(* IEC 61131-3 sources: elnaProjects/ElpcLogic/PomarKc7Changed/build_USO_ecl (part 8) *)

  IF isRunning THEN
  	Signaling := inSignaling;
  	SignalingTP := _signalingTp.Q;
  ELSE
  	Signaling := 0;
  	SignalingTP := 0;
  END_IF;

  IF NOT Remont AND NOT Check THEN
  	_signalingTp(in := Signaling, PT := T#1s);
  ELSE
  	_signalingTp(in := FALSE);
  END_IF;

  status :=  SHL(BYTE_TO_DWORD(source_for_Status), 29)
  			OR SHL(BYTE_TO_DWORD(cmd_for_Status), 26)
  			OR SHL(BYTE_TO_DWORD(command_error_for_Status), 23)
  			OR SHL(BOOL_TO_DWORD(OpcCommandsDisabled ), 21)
  			OR SHL(BOOL_TO_DWORD(Signaling), 16)
  			OR SHL(BOOL_TO_DWORD(RunOnStart ), 15)
  			OR SHL(BOOL_TO_DWORD(remont), 6)
  			OR SHL(BOOL_TO_DWORD(Check), 5)
  			OR SHL(BOOL_TO_DWORD(hasError), 4)
  			OR SHL(BOOL_TO_DWORD(SignalingTP), 3)
  			OR SHL(BOOL_TO_DWORD(CanRun), 2)
  			OR SHL(BOOL_TO_DWORD(isEnded), 1)
  			OR BOOL_TO_DWORD(isRunning);
END_FUNCTION_BLOCK

FUNCTION_BLOCK fb_BaseAlgoritm
  VAR_IN_OUT
    StrAlg : struct_Alg;
  END_VAR
  VAR
    _sunpackerCommand : fb_sunpackerCommand;
    source : BYTE;
    cmd : BYTE;
    lastCmd : BYTE;
    source_for_Status : BYTE;
    cmd_for_Status : BYTE;
    command_error_for_Status : BYTE;
    resetCmdTimer : TON;
    resetCmdTimerPriznak : BOOL;
  END_VAR

  StrAlg.CanRun := StrAlg.inCanRun;
  StrAlg.hasError := StrAlg.inHasError OR (command_error_for_Status <> 0);
  StrAlg.isEnded := StrAlg.inEnded;

  StrAlg.OpcCommandsDisabled := StrAlg.inOpcCommandsDisabled;

  (* ---- Если управление с ВУ заблокировано, то передаем команду из алгоритма ---- *)
  IF StrAlg.inOpcCommandsDisabled THEN
  	StrAlg.inCommand := StrAlg.inCommand_Alg;
  ELSE (* иначе передаем команду с АРМа*)
  	StrAlg.inCommand := StrAlg.inCommand_ARM;
  END_IF;

  _sunpackerCommand(command := StrAlg.inCommand);
  	source := _sunpackerCommand.source;
  	cmd := _sunpackerCommand.cmd;

  IF cmd <> 0 AND lastCmd <> cmd AND (((NOT StrAlg.opcCommandsDisabled) AND source > 0) OR source = 0) then
  	CASE BYTE_TO_INT(cmd) OF
  		(*cmdRun*) 1: 	IF (StrAlg.CanRun) THEN
  					StrAlg.isRuning := TRUE;
  					StrAlg.isEnded := FALSE;
  					StrAlg.hasError 	:= FALSE;

  					cmd_for_Status := cmd;
  					source_for_Status := source;
  					command_error_for_Status := 0;
  				ELSE
  					StrAlg.isRuning := FALSE;
  					StrAlg.isEnded := FALSE;
  					StrAlg.hasError 	:= FALSE;

  					cmd_for_Status := 0;
  					source_for_Status := source;
  					command_error_for_Status := cmd;
  				END_IF;
  		(*cmdReset*) 2: 	StrAlg.isRuning := FALSE;
  				StrAlg.isEnded := FALSE;
  				StrAlg.hasError 	:= FALSE;
  				cmd_for_Status := cmd;
  				source_for_Status := source;
  				command_error_for_Status := 0;
  	END_CASE;
  	resetCmdTimer(IN := false);
  	resetCmdTimerPriznak := TRUE;
  END_IF;
  lastCmd := cmd;

  resetCmdTimer(IN := resetCmdTimerPriznak, PT := T#5S);
  IF resetCmdTimer.Q THEN
  	resetCmdTimerPriznak := FALSE;
  	source_for_Status := 0;
  	cmd_for_Status := 0;
  	command_error_for_Status := 0;
  END_IF;

  StrAlg.status :=  SHL(BYTE_TO_DWORD(source_for_Status), 29)
  			OR SHL(BYTE_TO_DWORD(cmd_for_Status), 26)
  			OR SHL(BYTE_TO_DWORD(command_error_for_Status), 23)
  			OR SHL(BOOL_TO_DWORD(StrAlg.OpcCommandsDisabled ), 21)
  			OR SHL(BOOL_TO_DWORD(StrAlg.hasError),4)
  			OR SHL(BOOL_TO_DWORD(StrAlg.CanRun),2)
  			OR SHL(BOOL_TO_DWORD(StrAlg.isEnded),1)
  			OR BOOL_TO_DWORD(StrAlg.isRuning);
END_FUNCTION_BLOCK

FUNCTION_BLOCK fb_Switch
  VAR_INPUT
    statOn : BOOL;
    statOff : BOOL;
    statOn_reliability : BOOL;
    statOff_reliability : BOOL;
  END_VAR
  VAR_IN_OUT
    StrSw : struct_Switch;
  END_VAR
  VAR_INPUT
    inNs : TYPE_ReliableBit;
    inAccident : TYPE_ReliableBit;
    inAuto : TYPE_ReliableBit;
    inManual : TYPE_ReliableBit;
    inLocal : TYPE_ReliableBit;
    inDistance : TYPE_ReliableBit;
    inErrorPowerOff : TYPE_ReliableBit;
    inErrorBlock : TYPE_ReliableBit;
    inBreakCmdOn : TYPE_ReliableBit;
    inBreakCmdOff : TYPE_ReliableBit;
  END_VAR
  VAR
    onInit : BOOL          := FALSE;
    _statOn : BOOL;
    _statOff : BOOL;
    lastOnStatus : BYTE;
    cmd : BYTE;
    source : BYTE;
    lastCmd : BYTE;
    source_for_Status : BYTE;
    cmd_for_Status : BYTE;
    command_error_for_Status : BYTE;
    _sunpackerCommand : fb_sunpackerCommand;
    _statusDualInput : TYPE_statusDualInput;
    _commandDualInput : TYPE_commandDualInput;
    _commandErrorTimer : BOOL;
    resetErrorTimer : BOOL;
    getSdvig : BOOL;
    _changWithoutCommand : BOOL;
    errorCMDTimer : TON;
    sdvigReset : TON;
    _errorReset : TON;
    outputsSets : TOF;
  END_VAR
  VAR_IN_OUT
    cmdOn : BOOL;
    cmdOff : BOOL;
  END_VAR

  IF NOT onInit THEN
  IF StrSw.ISVALIDREF_cmdOn XOR StrSw.ISVALIDREF_cmdOff THEN
  	IF 	StrSw.ISVALIDREF_cmdOn THEN
  		lastCmd:= 2; (*baseCmdOff*)
  	ELSE
  		lastCmd:= 1; (*baseCmdOn*)
  	END_IF;
  END_IF;
  onInit:=TRUE;
  END_IF;

  (* ---- Если управление с ВУ заблокировано, то в ИМ передаем команду из алгоритма ---- *)
  IF StrSw.inOpcCommandsDisabled THEN
  	StrSw.inCommand := StrSw.inCommand_Alg;
  ELSE (* иначе передаем команду с АРМа*)
  	StrSw.inCommand := StrSw.inCommand_ARM;
  END_IF;

  (* ---- Формирование состояния механизма ---- *)

  IF (StrSw.ISVALIDREF_statOn) OR (StrSw.ISVALIDREF_statOff) THEN
  	IF (StrSw.ISVALIDREF_statOn) AND (StrSw.ISVALIDREF_statOff) THEN
  	StrSw.reliability:= statOn_reliability AND statOff_reliability;
  		_statOn  := statOn;
  		_statOff := statOff;
  	ELSIF (StrSw.ISVALIDREF_statOn) THEN
                       StrSw.reliability:= statOn_reliability;
  		_statOn  := statOn;
  		_statOff := NOT statOn;
  	ELSIF (StrSw.ISVALIDREF_statOff) THEN
  		 StrSw.reliability:= statOff_reliability;
  		_statOn  := NOT statOff;
  		_statOff :=statOff;
  	END_IF;

  	IF StrSw.reliability THEN
  		IF _statOn AND NOT _statOff 		THEN 	StrSw.onStatus := _statusDualInput.STATUS_ON;
  		ELSIF _statOff AND NOT _statOn 	THEN 	StrSw.onStatus := _statusDualInput.Status_OFF;
  		ELSIF NOT _statOn AND NOT _statOff 	THEN 	StrSw.onStatus := _statusDualInput.STATUS_TRANSITIONAL;
  		ELSE					StrSw.onStatus := _statusDualInput.STATUS_ERROR;
                      END_IF;

  	ELSE
  		StrSw.onStatus := _statusDualInput.STATUS_NOTDEFINED;

  	END_IF;
  ELSE
  	CASE BYTE_TO_INT(lastCmd) OF
  		(*baseCmdOn*) 1: StrSw.onStatus  := _statusDualInput.STATUS_ON;
  		(*baseCmdOff*) 2: StrSw.onStatus  := _statusDualInput.STATUS_OFF;

  	ELSE
  		 StrSw.onStatus := _statusDualInput.STATUS_NOTDEFINED;

  	END_CASE;
  END_IF;

  StrSw.Accident := inAccident.value AND inAccident.reliability;
  StrSw.Ns := inNs.value AND inNs.reliability;
  StrSw.Auto := inAuto.value AND inAuto.reliability;
  StrSw.Manual := inManual.value AND inManual.reliability;
  StrSw.Local := inLocal.value AND inLocal.reliability;
  StrSw.Distance := inDistance.value AND inDistance.reliability;
  StrSw.ErrorPowerOff := inErrorPowerOff.value AND inErrorPowerOff.reliability;
  StrSw.ErrorBlock := inErrorBlock.value AND inErrorBlock.reliability;
  StrSw.OpcCommandsDisabled := StrSw.inOpcCommandsDisabled;

  (* ---- Формирование признака сдвига ---- *)
  getSdvig := FALSE;
  IF (StrSw.ISVALIDREF_cmdOn OR StrSw.ISVALIDREF_cmdOff) AND NOT StrSw.Local THEN
  	IF NOT (StrSw.CmdOn OR StrSw.CmdOff) THEN
                       IF (lastOnStatus <> StrSw.onStatus AND
  		(StrSw.onStatus <> _statusDualInput.STATUS_NOTDEFINED AND
                       StrSw.onStatus <> _statusDualInput.STATUS_ERROR)     AND
  		(lastOnStatus <> _statusDualInput.STATUS_NOTDEFINED   AND
                       lastOnStatus <> _statusDualInput.STATUS_ERROR))
                      THEN
  			getSdvig   := TRUE;
  		END_IF;
  	END_IF;
  END_IF;

  IF getSdvig THEN StrSw.sdvig:= TRUE; END_IF;

  sdvigReset(IN:=StrSw.sdvig, PT:=T#15S);

  IF sdvigReset.Q THEN StrSw.sdvig:=FALSE; END_IF;

  lastOnStatus := StrSw.onStatus;

  (* ---- Распаковка команды ---- *)
  _sunpackerCommand(command := StrSw.inCommand);
  	cmd := _sunpackerCommand.cmd;
  	source := _sunpackerCommand.source;

  (* ---- Обработка команды ---- *)
  IF cmd <> 0 AND lastCmd <> cmd and (((NOT StrSw.opcCommandsDisabled) AND source > 0) OR source = 0) then
  	CASE BYTE_TO_INT(cmd) OF
  	(*cmd_open*) 1 :
  			IF  StrSw.ISVALIDREF_cmdOn THEN StrSw.CmdOn := TRUE;
  				IF StrSw.ISVALIDREF_cmdOff THEN StrSw.CmdOff := FALSE; END_IF;
  			ELSIF  StrSw.ISVALIDREF_cmdOff THEN StrSw.CmdOff := FALSE;  END_IF;
                                lastCmd := cmd;
  			errorCMDTimer(IN := false);
  			_commandErrorTimer := true;
  			StrSw.lastCmdIsOn := true;
  	(*cmd_close*) 2 :
  			IF StrSw.ISVALIDREF_cmdOff THEN StrSw.CmdOff := TRUE;
  				IF StrSw.ISVALIDREF_cmdOn THEN StrSw.CmdOn := FALSE; END_IF;
  			ELSIF StrSw.ISVALIDREF_cmdOn THEN StrSw.CmdOn := FALSE; END_IF;
                                lastCmd := cmd;
  			errorCMDTimer(IN := false);
  			_commandErrorTimer := true;
  			StrSw.lastCmdIsOn := false;
  	(*cmd_reset*) 3 :    IF StrSw.ISVALIDREF_statOn OR StrSw.ISVALIDREF_statOff THEN
  			StrSw.CmdOn := FALSE;
  			StrSw.CmdOff := FALSE;
                                lastCmd :=0;
  			_commandErrorTimer := false;
  			StrSw.lastCmdIsOn := false;
                                 END_IF;
  	END_CASE;
  	source_for_Status := source;
  	cmd_for_Status := cmd;
  	command_error_for_Status := 0;
  END_IF;

  errorCMDTimer(In := _commandErrorTimer, PT :=T#10s);

  (* ---- алгоритм  для команды ВКЛючить ---- *)
  IF (StrSw.onStatus = _statusDualInput.STATUS_ON) and StrSw.lastCmdIsOn then
  	IF StrSw.ISVALIDREF_cmdOn AND StrSw.ISVALIDREF_cmdOff then  StrSw.cmdOn := false; END_IF;

  	 errorCMDTimer(In := false);
  	 _commandErrorTimer := false;
  	 cmd_for_Status := 0;
  	 source_for_Status := 0;
  END_IF;

  (* ---- off ---- *)
  IF (StrSw.onStatus = _statusDualInput.STATUS_OFF) and (NOT StrSw.lastCmdIsOn) then
  	IF StrSw.ISVALIDREF_cmdOn AND StrSw.ISVALIDREF_cmdOff then  StrSw.cmdOff := false; END_IF;

  	 errorCMDTimer(In := false);
  	 _commandErrorTimer := false;
  	 cmd_for_Status := 0;
  	 source_for_Status := 0;
  END_IF;

  (* ---- ошибка исполнения команды ---- *)
  if errorCMDTimer.Q and (cmd_for_Status <> 0) then
  	command_error_for_Status :=  cmd_for_Status;
  	_commandErrorTimer := false;
  	StrSw.CmdOn := false;
  	StrSw.CmdOff := false;
  	lastCmd := 0;
  end_if;

  (* ---- сброс ошибки команды ---- *)
  StrSw.CommandFault := command_error_for_Status <> 0;
  _errorReset(IN := command_error_for_Status <> 0, PT := T#5S);
  IF _errorReset.Q THEN
  	cmd_for_Status := 0;
  	source_for_Status := 0;
  	command_error_for_Status := 0;
  END_IF;

  outputsSets(in := (StrSw.ISVALIDREF_cmdOn and StrSw.cmdOn ) OR (StrSw.ISVALIDREF_cmdOff and StrSw.cmdOff), PT := T#2S);
  	IF NOT outputsSets.Q THEN
  		StrSw.BreakCmdOn := inBreakCmdOn._inversed AND
                      inBreakCmdOn.reliability AND StrSw.ISVALIDREF_inBreakCmdOn;

  		StrSw.BreakCmdOff := inBreakCmdOff._inversed
                      AND inBreakCmdOff.reliability AND StrSw.ISVALIDREF_inBreakCmdOff;
  	END_IF;

  cmdOn := StrSw.cmdOn;
  cmdOff:= StrSw.cmdOff;

  (* ---- формирование зашифрованного статуса для АРМа ---- *)
  StrSw.status := shl(BYTE_TO_DWORD(source_for_Status), 29)
  		OR shl(BYTE_TO_DWORD(cmd_for_Status), 26)
  		OR shl(BYTE_TO_DWORD(command_error_for_Status), 23)
  		OR shl(bool_to_DWORD(StrSw.sdvig), 22)
  		OR shl(bool_to_DWORD(StrSw.OpcCommandsDisabled), 21)
                      OR shl(bool_to_DWORD(StrSw.lastCmdIsOn), 14)
                      OR shl(BOOL_TO_DWORD(StrSw.BreakCmdOff), 13)
  		OR shl(BOOL_TO_DWORD(StrSw.BreakCmdOn), 12)
  		OR shl(BOOL_TO_DWORD(StrSw.ErrorBlock), 11)
  		OR shl(BOOL_TO_DWORD(StrSw.ErrorPowerOff), 10)
  		OR shl(BOOL_TO_DWORD(StrSw.Manual), 8)
  		OR shl(BOOL_TO_DWORD(StrSw.Auto), 7)
  		OR shl(BOOL_TO_DWORD(StrSw.Distance), 6)
  		OR shl(BOOL_TO_DWORD(StrSw.Local), 5)
  		OR shl(BOOL_TO_DWORD(StrSw.Ns), 4)
                  	OR shl(BOOL_TO_DWORD(StrSw.Accident ),3)
  		OR BYTE_TO_DWORD(StrSw.onStatus);
END_FUNCTION_BLOCK

FUNCTION_BLOCK fb_singleOutput
  VAR_IN_OUT
    signal : BOOL;
    str_SO : struct_singleOutput;
  END_VAR
  VAR
    pulseTimer : TON;
    resetCmdTimer : TON;
    TON_Command : TON;
    source : BYTE;
    cmd : BYTE;
    lastCmd : BYTE;
    source_for_Status : BYTE;
    cmd_for_Status : BYTE;
    command_error_for_Status : BYTE;
    pulseTimerPriznak : BOOL;
    resetCmdTimerPriznak : BOOL;
    _sunpackerCommand : fb_sunpackerCommand;
  END_VAR

  str_SO.OpcCommandsDisabled := str_SO.inOpcCommandsDisabled;

  (* ---- Если управление с ВУ заблокировано, то передаем команду из алгоритма ---- *)
  IF str_SO.inOpcCommandsDisabled THEN
  	str_SO.inCommand := str_SO.inCommand_Alg;
  ELSE (* иначе передаем команду с АРМа*)
  	str_SO.inCommand := str_SO.inCommand_ARM;
  END_IF;

  (*Распаковка команды*)
  _sunpackerCommand(command := str_SO.inCommand);
  	cmd := _sunpackerCommand.cmd;
  	source := _sunpackerCommand.source;

  (*Обработка команды*)
  IF cmd <> 0 AND lastCmd <> cmd and (((NOT str_SO.OpcCommandsDisabled) AND source > 0) OR source = 0) then
  	CASE BYTE_TO_INT(cmd) OF
  	(*cmd_on*) 1 :
  			str_SO.Q := TRUE;
  			pulseTimer(IN := FALSE);
  			pulseTimerPriznak := FALSE;
  			resetCmdTimer(IN := FALSE);
  			resetCmdTimerPriznak := TRUE;
  	(*cmd_off*) 2 :
  			str_SO.Q := FALSE;
  			pulseTimer(IN := FALSE);
  			pulseTimerPriznak := FALSE;
  			resetCmdTimer(IN := FALSE);
  			resetCmdTimerPriznak := TRUE;
  	(*cmd_pulse*) 3 :
  			str_SO.Q := TRUE;
                                pulseTimer(IN := FALSE);
                                pulseTimerPriznak := TRUE;
  			resetCmdTimer(IN := FALSE);
                                resetCmdTimerPriznak := FALSE;
  	END_CASE;
  	source_for_Status := source;
  	cmd_for_Status := cmd;
  	command_error_for_Status := 0;
  END_IF;
  lastCmd := cmd;

  pulseTimer(IN := pulseTimerPriznak, PT := str_SO.wait_time);
  pulseTimer();
  IF pulseTimer.Q THEN
  	pulseTimer(IN := FALSE);
  	pulseTimerPriznak := FALSE;

  	str_SO.Q := FALSE;

  	source_for_Status := 0;
  	cmd_for_Status := 0;
  	command_error_for_Status := 0;
  END_IF;

  resetCmdTimer(IN := resetCmdTimerPriznak, PT := T#10S);
  resetCmdTimer();
  IF resetCmdTimer.Q THEN
  	resetCmdTimer(IN := FALSE);
  	resetCmdTimerPriznak := FALSE;

  	source_for_Status := 0;
  	cmd_for_Status := 0;
  	command_error_for_Status := 0;
  END_IF;

  signal:= str_SO.Q;

  (*TON_Command(IN:= (inCommand <> 0) AND (source = 0), PT:= T#2S);*)
      (*IF TON_Command.Q THEN*)
          (*inCommand := 0;*)
      (*END_IF;*)
  str_SO.status :=                           shl(BYTE_TO_DWORD(source_for_Status), 29)
  				OR shl(BYTE_TO_DWORD(cmd_for_Status), 26)
  				OR shl(BYTE_TO_DWORD(command_error_for_Status), 23)
  				OR shl(BOOL_TO_DWORD(str_SO.OpcCommandsDisabled), 21)
  				OR BOOL_TO_DWORD(str_SO.Q);
END_FUNCTION_BLOCK

FUNCTION_BLOCK proc_IM
  VAR
    fb_Kran1 : fb_Kran;
    fb_Kran2 : fb_Kran;
    fb_Kran3 : fb_Kran;
    fb_Kran3b : fb_Kran;
    fb_Kran4 : fb_Kran;
    fb_Kran5 : fb_Kran;
    fb_Kran6 : fb_Kran;
    fb_nu1 : fb_OilPump;
    fb_nu2 : fb_OilPump;
    fb_pns : fb_Switch;
    fb_v1_Avom : fb_Switch;
    fb_v2_Avom : fb_Switch;
    fb_v3_Avom : fb_Switch;
    fb_v4_Avom : fb_Switch;
    fb_TEN_kollectora : fb_Switch;
    fb_KaloriferAVOM : fb_Switch;
    fb_CMN : fb_Switch;
    fb_TEN_MB : fb_Switch;
    fb_mv : fb_SectionSwitch;
    fb_PLC_Control : fb_meandr;
  END_VAR
  VAR_EXTERNAL
    di : DiConfig;
    od : DOconfig;
    IM : ImConfig;
  END_VAR
  VAR
    fb_dP_maslo_gaz_Less100 : fb_singleSignal;
    fb_dp_kran1_Less100 : fb_singleSignal;
    fb_QF1_on : fb_singleSignal;
    fb_QF2_on : fb_singleSignal;
    fb_QF23_on : fb_singleSignal;
    fb_QF4_QF5_on : fb_singleSignal;
    fb_QF6_QF7_on : fb_singleSignal;
    fb_QF8_QF9_on : fb_singleSignal;
    fb_QF10_QF11_on : fb_singleSignal;
    fb_QF12_QF13_on : fb_singleSignal;
    fb_QF14_QF15_on : fb_singleSignal;
    fb_QF22_on : fb_singleSignal;
    fb_NS_G1_G2 : fb_singleSignal;
    fb_NS_G3_G4 : fb_singleSignal;
    fb_NS_G15_G16 : fb_singleSignal;
    fb_NS_G17 : fb_singleSignal;
    fb_NS_G5_G6 : fb_singleSignal;
    fb_NS_G7_G8 : fb_singleSignal;
    fb_NS_G18_G19 : fb_singleSignal;
    fb_NS_G10_G11 : fb_singleSignal;
    fb_NS_G13_G14 : fb_singleSignal;
    fb_Vozbud_neispr_tsepey_upr_AVR_pit : fb_singleSignal;
    fb_Vozbud_gotovnost : fb_singleSignal;
    fb_Vozbud_neispravnost : fb_singleSignal;
    fb_SHAVR1_v_rabote : fb_singleSignal;
    fb_SHAVR2_v_rabote : fb_singleSignal;
    fb_Avariinoe_otkluch_vikluchatelya : fb_singleSignal;
    fb_Assinhronnii_hod_peregruzka : fb_singleSignal;
    fb_SHU_v_GPA_vkluch : fb_singleSignal;
    fb_SHP_v_GPA_vkluch : fb_singleSignal;
    fb_Uroven_masla_akkum : fb_singleSignal;
    fb_NKU1_GPA_on : fb_singleSignal;
    fb_NKU2_GPA_on : fb_singleSignal;
    fb_AO_KC_ot_SHKS : fb_singleSignal;
    fb_AO_GPA_ot_SHU : fb_singleSignal;
    fb_BEAO_srabotal : fb_singleSignal;
    fb_Chastotny_pusk : fb_singleSignal;
    fb_Neuspesh_chastotny_pusk : fb_singleSignal;
    fb_Rezhim_ruchnogo_regulirovaniya : fb_singleSignal;
    fb_Razreshenie_zagruzki_dvig : fb_singleSignal;
    fb_Osnovnoy_regul_off : fb_singleSignal;
    fb_Voltage_sekcii_norm : fb_singleSignal;
    fb_Reactorny_pusk : fb_singleSignal;
    fb_NO_GPA_ot_SHU : fb_singleSignal;
    fb_AO_GPA_ot_PRU : fb_singleSignal;
    fb_Nalichie_BP1 : fb_singleSignal;
    fb_Nalichie_BP2 : fb_singleSignal;
    fb_Nalichie_BP3 : fb_singleSignal;
    fb_Nalichie_BP4 : fb_singleSignal;
    fb_Nalichie_BP5 : fb_singleSignal;
    fb_Nalichie_BP6 : fb_singleSignal;
    fb_Nalichie_BP7_BP8 : fb_singleSignal;
    fb_Nalichie_BP9_BP10 : fb_singleSignal;
    fb_Nalichie_cepei_upravlen_mv : fb_singleSignal;
    fb_Nalichie_220BEAO : fb_singleSignal;
    fb_Nalichie_per_220_na_vhode : fb_singleSignal;
    fb_Nalichie_post_220_na_vhode : fb_singleSignal;
    fb_Nalichie_BP11 : fb_singleSignal;
    fb_Nalichie_BP12 : fb_singleSignal;
    fb_Dver_SHU_pered_otkrita : fb_singleSignal;
    fb_Dver_SHU_zad_otkrita : fb_singleSignal;
    fb_EO_GPA_ot_knopki_SHU : fb_singleSignal;
    fb_EO_EGPA_ot_PRY : fb_singleSignal;
    fb_Synchroniz_rezhima_K1 : fb_singleSignal;
    fb_Potok_ms_posle_AVOM : fb_singleSignal;
    fb_Avary_EGPA : fb_singleOutput;
    fb_U_lamp_SHU : fb_singleOutput;
    fb_AO_knopka_ind : fb_singleOutput;
    fb_Pusk : fb_singleOutput;
    fb_Stop_SHUP : fb_singleOutput;
    fb_NO_fonar : fb_singleOutput;
    fb_PC_fonar : fb_singleOutput;
    fb_AC_fonar : fb_singleOutput;
    fb_Kr1_smazka : fb_singleOutput;
    fb_Kr2_smazka : fb_singleOutput;
    fb_Kr4_open_from_alg : fb_singleOutput;
    fb_Synch_rej_K1 : fb_singleOutput;
    fb_Rabota_EGPA : fb_singleOutput;
    fb_Neispr_EGPA : fb_singleOutput;
  END_VAR

  (* Циклический опрос. ИМ *)

  (* GPIO *)
  fb_PLC_Control(output:=od.gpio_out.bits[0]);

  (* Кран 1 *)
  fb_Kran1(statOn := di.di_20.bits[5]._inversed,
           statOff := di.di_20.bits[4]._inversed,
           inSo := di.di_16.bits[0], inSz := di.di_16.bits[1],
           cmdOn:=od.do_0.bits[0], cmdOff:=od.do_0.bits[1],
           strKr:= IM.Kran1  );

  (* Кран 2 *)
  fb_Kran2(statOn := di.di_21.bits[0]._inversed,
           statOff := di.di_20.bits[7]._inversed,
           inSo := di.di_16.bits[2], inSz := di.di_16.bits[3],
           cmdOn:=od.do_0.bits[2], cmdOff:=od.do_0.bits[3],
           strKr:= IM.Kran2  );

  (* Кран 3 *)
  fb_Kran3(statOn := di.di_0.bits[5]._inversed,
           statOff := di.di_0.bits[4]._inversed,
           inSo := di.di_16.bits[4], inSz := di.di_16.bits[5],
           cmdOn:=od.do_0.bits[4], cmdOff:=od.do_0.bits[5],
           strKr:= IM.Kran3  );

  (* Кран 3b *)
  fb_Kran3b(statOn := di.di_0.bits[7]._inversed,
           statOff := di.di_0.bits[6]._inversed,
           inSo := di.di_16.bits[6], inSz := di.di_16.bits[7],
           cmdOn:=od.do_0.bits[6], cmdOff:=od.do_0.bits[7],
           strKr:= IM.Kran3b  );

  (* Кран 4 *)
  fb_Kran4(statOn := di.di_1.bits[1]._inversed,
           statOff := di.di_1.bits[0]._inversed,
           inSo := di.di_17.bits[0], inSz := di.di_17.bits[1],
           cmdOn:=od.do_0.bits[8], cmdOff:=od.do_0.bits[9],
           strKr:= IM.Kran4  );

  (* Кран 5 *)
  fb_Kran5(statOn := di.di_1.bits[3]._inversed,
           statOff := di.di_1.bits[2]._inversed,
           inSo := di.di_17.bits[2], inSz := di.di_17.bits[3],
           cmdOn:=od.do_0.bits[10], cmdOff:=od.do_0.bits[11],
           strKr:= IM.Kran5  );

  (* Кран 6НР *)
  fb_Kran6(statOn := di.di_1.bits[5]._inversed,
           statOff := di.di_1.bits[4]._inversed,
           inSo := di.di_17.bits[4], inSz := di.di_17.bits[5],
           cmdOn:=od.do_0.bits[12], cmdOff:=od.do_0.bits[13],
           strKr:= IM.Kran6  );

  (*  НУ1 Насос уплотнения *)
  fb_nu1(statOn := di.di_5.bits[1].value, statOff := di.di_5.bits[1]._inversed,
           cmdOn:=od.do_1.bits[4], cmdOff:=od.do_1.bits[5],
           StrSw:= IM.nu1  );

  (*  НУ2 Насос уплотнения *)
  fb_nu2(statOn := di.di_5.bits[2].value, statOff := di.di_5.bits[2]._inversed,
           cmdOn:=od.do_1.bits[6], cmdOff:=od.do_1.bits[7],
           StrSw:= IM.nu2  );

  (*  ПНС Насос смазки *)
  fb_pns(statOn := di.di_5.bits[0].value, statOff := di.di_5.bits[0]._inversed,
           cmdOn:=od.do_1.bits[0], cmdOff:=od.do_1.bits[1],
           StrSw:= IM.pns  );

  (*  В1 АВОМ вентилятор охлаждения *)
  fb_v1_Avom(statOn := di.di_5.bits[3].value, statOff := di.di_5.bits[3]._inversed,
           cmdOn:=od.do_1.bits[8], cmdOff:=od.do_1.bits[9],
           StrSw:= IM.v1_Avom  );

  (*  В2 АВОМ вентилятор охлаждения *)
  fb_v2_Avom(statOn := di.di_5.bits[4].value, statOff := di.di_5.bits[4]._inversed,
           cmdOn:=od.do_1.bits[10], cmdOff:=od.do_1.bits[11],
           StrSw:= IM.v2_Avom  );

  (*  В3 АВОМ вентилятор охлаждения *)
  fb_v3_Avom(statOn := di.di_5.bits[5].value, statOff := di.di_5.bits[5]._inversed,
           cmdOn:=od.do_1.bits[12], cmdOff:=od.do_1.bits[13],
           StrSw:= IM.v3_Avom  );

  (*  В4 АВОМ вентилятор охлаждения *)
  fb_v4_Avom(statOn := di.di_5.bits[6].value, statOff := di.di_5.bits[6]._inversed,
           cmdOn:=od.do_1.bits[14], cmdOff:=od.do_1.bits[15],
           StrSw:= IM.v4_Avom  );

  (*  МВ масляный выключатель *)
  fb_mv(statOn := di.di_7.bits[0].value, statOff := di.di_20.bits[3].value,
           basketRolledin:= di.di_7.bits[2], basketRolledout:= di.di_7.bits[2],
           cmdOn:=od.do_4.bits[6] , cmdOff:=od.do_4.bits[7],
           StrSw:= IM.mv  );

  (* Тен коллектора *)
  fb_TEN_kollectora(statOn := di.di_10.bits[1].value, statOff := di.di_10.bits[1]._inversed,
           cmdOn:=od.do_2.bits[6], cmdOff:=od.do_2.bits[6],
           StrSw:= IM.TEN_kollectora  );

  (* Калорифер АВОМ *)
  fb_KaloriferAVOM(statOn := di.di_10.bits[2].value, statOff := di.di_10.bits[2]._inversed,
           cmdOn:=od.do_2.bits[0], cmdOff:=od.do_2.bits[1],
           StrSw:= IM.KaloriferAVOM  );

  (* ЦМН *)
  fb_CMN(statOn := di.di_10.bits[3].value, statOff := di.di_10.bits[3]._inversed,
           cmdOn:=od.do_2.bits[4], cmdOff:=od.do_2.bits[5],
           StrSw:= IM.CMN);

  (* Тен маслобака *)
  fb_TEN_MB(statOn := di.di_10.bits[0].value, statOff := di.di_10.bits[0]._inversed,
           cmdOn:=od.do_2.bits[2], cmdOff:=od.do_2.bits[3],
           StrSw:= IM.TEN_MB);
  (*************************************************** singleSignals ********************************************)

  (* Перепад давления масло газ м*)
  fb_dP_maslo_gaz_Less100(signal :=di.di_20.bits[6], str_SS := IM.SingleSignals.dP_maslo_gaz_Less100);

  (* Перепад давления кран 1 *)
  fb_dp_kran1_Less100(signal :=di.di_4.bits[1], str_SS := IM.SingleSignals.dp_kran1_Less100);

  (* Неисправность цепей управления возбудителя *)
  fb_Vozbud_neispr_tsepey_upr_AVR_pit(signal :=di.di_6.bits[4], str_SS := IM.SingleSignals.Vozbud_neispr_tsepey_upr_AVR_pit);

  (* Возбудитель готовность *)
  fb_Vozbud_gotovnost(signal :=di.di_6.bits[0], str_SS := IM.SingleSignals.Vozbud_gotovnost);

  (* Возбудитель неисправность *)
  fb_Vozbud_neispravnost(signal :=di.di_21.bits[7], str_SS := IM.SingleSignals.Vozbud_neispravnost);

  (* ЩАВР 1 в работе *)
  fb_SHAVR1_v_rabote(signal :=di.di_13.bits[6], str_SS := IM.SingleSignals.SHAVR1_v_rabote);

  (* ЩАВР 2 в работе *)
  fb_SHAVR2_v_rabote(signal :=di.di_13.bits[7], str_SS := IM.SingleSignals.SHAVR2_v_rabote);

  (* ЩАВР 2 в работе *)
  fb_Avariinoe_otkluch_vikluchatelya(signal :=di.di_8.bits[0], str_SS := IM.SingleSignals.Avariinoe_otkluch_vikluchatelya);

  (* ЩАВР 2 в работе *)
  fb_Assinhronnii_hod_peregruzka(signal :=di.di_8.bits[1], str_SS := IM.SingleSignals.Assinhronnii_hod_peregruzka);

  (* ЩАВР 2 в работе *)
  fb_SHU_v_GPA_vkluch(signal :=di.di_8.bits[2], str_SS := IM.SingleSignals.SHU_v_GPA_vkluch);

  (* ЩАВР 2 в работе *)
  fb_SHP_v_GPA_vkluch(signal :=di.di_8.bits[3], str_SS := IM.SingleSignals.SHP_v_GPA_vkluch);

  (* ЩАВР 2 в работе *)
  fb_Uroven_masla_akkum(signal :=di.di_4.bits[2], str_SS := IM.SingleSignals.Uroven_masla_akkum);

  (* ЩАВР 2 в работе *)
  fb_NKU1_GPA_on(signal :=di.di_10.bits[4], str_SS := IM.SingleSignals.NKU1_GPA_on);

  (* ЩАВР 2 в работе *)
  fb_NKU2_GPA_on(signal :=di.di_10.bits[5], str_SS := IM.SingleSignals.NKU2_GPA_on);

  (* ЩАВР 2 в работе *)
  fb_AO_KC_ot_SHKS(signal :=di.di_20.bits[0], str_SS := IM.SingleSignals.AO_KC_ot_SHKS);

  (* ЩАВР 2 в работе *)
  fb_AO_GPA_ot_SHU(signal :=di.di_21.bits[2], str_SS := IM.SingleSignals.AO_GPA_ot_SHU);

  (* ЩАВР 2 в работе *)
  fb_BEAO_srabotal(signal :=di.di_18.bits[1], str_SS := IM.SingleSignals.BEAO_srabotal);

  (* ЩАВР 2 в работе *)
  fb_Chastotny_pusk(signal :=di.di_9.bits[0], str_SS := IM.SingleSignals.Chastotny_pusk);

  (* ЩАВР 2 в работе *)
  fb_Neuspesh_chastotny_pusk(signal :=di.di_9.bits[1], str_SS := IM.SingleSignals.Neuspesh_chastotny_pusk);

  (* ЩАВР 2 в работе *)
  fb_Rezhim_ruchnogo_regulirovaniya(signal :=di.di_9.bits[2], str_SS := IM.SingleSignals.Rezhim_ruchnogo_regulirovaniya);

  (* ЩАВР 2 в работе *)
  fb_Razreshenie_zagruzki_dvig(signal :=di.di_6.bits[1], str_SS := IM.SingleSignals.Razreshenie_zagruzki_dvig);

  (* ЩАВР 2 в работе *)
  fb_Osnovnoy_regul_off(signal :=di.di_6.bits[3], str_SS := IM.SingleSignals.Osnovnoy_regul_off);

  (* ЩАВР 2 в работе *)
  fb_Voltage_sekcii_norm(signal :=di.di_8.bits[4], str_SS := IM.SingleSignals.Voltage_sekcii_norm);

  (* ЩАВР 2 в работе *)
  fb_Reactorny_pusk(signal :=di.di_8.bits[5], str_SS := IM.SingleSignals.Reactorny_pusk);

  (* ЩАВР 2 в работе *)
  fb_NO_GPA_ot_SHU(signal :=di.di_21.bits[1], str_SS := IM.SingleSignals.NO_GPA_ot_SHU);

  (* ЩАВР 2 в работе *)
  fb_AO_GPA_ot_PRU(signal :=di.di_21.bits[3], str_SS := IM.SingleSignals.AO_GPA_ot_PRU);

  (* ЩАВР 2 в работе *)
  fb_Nalichie_BP1(signal :=di.di_11.bits[0], str_SS := IM.SingleSignals.Nalichie_BP1);

  (* ЩАВР 2 в работе *)
  fb_Nalichie_BP2(signal :=di.di_11.bits[1], str_SS := IM.SingleSignals.Nalichie_BP2);

  (* ЩАВР 2 в работе *)
  fb_Nalichie_BP3(signal :=di.di_11.bits[2], str_SS := IM.SingleSignals.Nalichie_BP3);

  (* ЩАВР 2 в работе *)
  fb_Nalichie_BP4(signal :=di.di_11.bits[3], str_SS := IM.SingleSignals.Nalichie_BP4);

  (* ЩАВР 2 в работе *)
  fb_Nalichie_BP5(signal :=di.di_11.bits[4], str_SS := IM.SingleSignals.Nalichie_BP5);

  (* ЩАВР 2 в работе *)
  fb_Nalichie_BP6(signal :=di.di_11.bits[5], str_SS := IM.SingleSignals.Nalichie_BP6);

  (* ЩАВР 2 в работе *)
  fb_Nalichie_BP7_BP8(signal :=di.di_11.bits[6], str_SS := IM.SingleSignals.Nalichie_BP7_BP8);

  (* ЩАВР 2 в работе *)
  fb_Nalichie_BP9_BP10(signal :=di.di_11.bits[7], str_SS := IM.SingleSignals.Nalichie_BP9_BP10);

  (* ЩАВР 2 в работе *)
  fb_Nalichie_cepei_upravlen_mv(signal :=di.di_12.bits[0], str_SS := IM.SingleSignals.Nalichie_cepei_upravlen_mv);

  (* ЩАВР 2 в работе *)
  fb_Nalichie_220BEAO(signal :=di.di_12.bits[1], str_SS := IM.SingleSignals.Nalichie_220BEAO);

  (* ЩАВР 2 в работе *)
  fb_Nalichie_per_220_na_vhode(signal :=di.di_12.bits[2], str_SS := IM.SingleSignals.Nalichie_per_220_na_vhode);

  (* ЩАВР 2 в работе *)
  fb_Nalichie_post_220_na_vhode(signal :=di.di_12.bits[3], str_SS := IM.SingleSignals.Nalichie_post_220_na_vhode);

  (* ЩАВР 2 в работе *)
  fb_Nalichie_BP11(signal :=di.di_12.bits[4], str_SS := IM.SingleSignals.Nalichie_BP11);

  (* ЩАВР 2 в работе *)
  fb_Nalichie_BP12(signal :=di.di_12.bits[4], str_SS := IM.SingleSignals.Nalichie_BP12);

  (* ЩАВР 2 в работе *)
  fb_Dver_SHU_pered_otkrita(signal :=di.di_13.bits[0], str_SS := IM.SingleSignals.Dver_SHU_pered_otkrita);

  (* ЩАВР 2 в работе *)
  fb_Dver_SHU_zad_otkrita(signal :=di.di_13.bits[1], str_SS := IM.SingleSignals.Dver_SHU_zad_otkrita);

  (* ЩАВР 2 в работе *)
  fb_EO_GPA_ot_knopki_SHU(signal :=di.di_14.bits[0], str_SS := IM.SingleSignals.EO_GPA_ot_knopki_SHU);

  (* ЩАВР 2 в работе *)
  fb_EO_EGPA_ot_PRY(signal :=di.di_14.bits[1], str_SS := IM.SingleSignals.EO_EGPA_ot_PRY);

  (* ЩАВР 2 в работе *)
  fb_Synchroniz_rezhima_K1(signal :=di.di_3.bits[4], str_SS := IM.SingleSignals.Synchroniz_rezhima_K1);

  (* ЩАВР 2 в работе *)
  fb_Potok_ms_posle_AVOM(signal :=di.di_3.bits[4], str_SS := IM.SingleSignals.Potok_ms_posle_AVOM);

    (* Выключатель основного ввода питания QF1  в положении включен   *)
  fb_QF1_on(signal :=di.di_7.bits[6], str_SS := IM.SingleSignals.QF1_on);

    (* Выключатель резервного ввода питания QF2  в положении включен   *)
  fb_QF2_on(signal :=di.di_7.bits[7], str_SS := IM.SingleSignals.QF2_on);

    (* Выключатель питания кранов:  QF23 110 В в положении включен   *)
  fb_QF23_on(signal :=di.di_8.bits[0], str_SS := IM.SingleSignals.QF23_on);

    (* Выключатели группы 1: QF4, QF5 в положении включен   *)
  fb_QF4_QF5_on(signal :=di.di_8.bits[1], str_SS := IM.SingleSignals.QF4_QF5_on);

    (* Выключатели группы 2: QF6, QF7 в положении включен   *)
  fb_QF6_QF7_on(signal :=di.di_8.bits[2], str_SS := IM.SingleSignals.QF6_QF7_on);

    (* Выключатели группы 3: QF8, QF9 в положении включен   *)
  fb_QF8_QF9_on(signal :=di.di_8.bits[3], str_SS := IM.SingleSignals.QF8_QF9_on);

    (* Выключатели группы 4: QF10, QF11 в положении включен   *)
  fb_QF10_QF11_on(signal :=di.di_8.bits[4], str_SS := IM.SingleSignals.QF10_QF11_on);

    (* Выключатели группы 5: QF12, QF13 в положении включен   *)
  fb_QF12_QF13_on(signal :=di.di_8.bits[5], str_SS := IM.SingleSignals.QF12_QF13_on);

    (* Выключатели группы 6: QF14, QF15 в положении включен   *)
  fb_QF14_QF15_on(signal :=di.di_8.bits[6], str_SS := IM.SingleSignals.QF14_QF15_on);

    (* Выключатели группы : QF22 в положении включен   *)
  fb_QF22_on(signal :=di.di_14.bits[2], str_SS := IM.SingleSignals.QF22_on);

    (* Неисправность источников питания группы 1: G1, G2 (=24 В)   *)
  fb_NS_G1_G2(signal :=di.di_8.bits[7], str_SS := IM.SingleSignals.NS_G1_G2);

    (* Неисправность источников питания группы 2: G3, G4 (=24 В)   *)
  fb_NS_G3_G4(signal :=di.di_9.bits[0], str_SS := IM.SingleSignals.NS_G3_G4);

    (* Неисправность источников питания внутренних ПТС: G15, G16 (=24 В)   *)
  fb_NS_G15_G16(signal :=di.di_9.bits[1], str_SS := IM.SingleSignals.NS_G15_G16);

    (* Неисправность источника питания аналоговых сигналов: G17 (=24 В)   *)
  fb_NS_G17(signal :=di.di_9.bits[2], str_SS := IM.SingleSignals.NS_G17);

    (* Неисправность источников питания группы 3: G5, G6 (=24 В)   *)
  fb_NS_G5_G6(signal :=di.di_9.bits[3], str_SS := IM.SingleSignals.NS_G5_G6);

    (* Неисправность источников питания группы 4: G7, G8 (=24 В)   *)
  fb_NS_G7_G8(signal :=di.di_9.bits[4], str_SS := IM.SingleSignals.NS_G7_G8);

    (* Неисправность источников питания внешних цепей: G18, G19 (=24 В)   *)
  fb_NS_G18_G19(signal :=di.di_9.bits[5], str_SS := IM.SingleSignals.NS_G18_G19);

    (* Неисправность источников питания группы 5: G9, G10, G11, G12 (=110 В)   *)
  fb_NS_G10_G11(signal :=di.di_9.bits[6], str_SS := IM.SingleSignals.NS_G10_G11);

    (* Неисправность источников питания G13, G14 (=24 В)   *)
  fb_NS_G13_G14(signal :=di.di_9.bits[7], str_SS := IM.SingleSignals.NS_G13_G14);

  (*************************************************** SingleOutputs ********************************************)

  (* Идикация НО (подсветка кнопки на шкафу)   *)
  fb_Rabota_EGPA(str_SO := IM.SingleOutputs.Rabota_EGPA, signal:=od.do_4.bits[2]);

  (* Взвод включения БЭАО по неисправности ПТС   *)
  fb_Neispr_EGPA(str_SO := IM.SingleOutputs.Neispr_EGPA, signal:=od.do_4.bits[0]);

  (* Авария ЭГПА в КЦ
  fb_Avary_EGPA(str_SO := IM.SingleOutputs.Avary_EGPA, signal:=od.do_4.bits[1);  *)

  (* Сброс включения БЭАО по неисправности ПТС   *)
  fb_U_lamp_SHU(str_SO := IM.SingleOutputs.U_lamp_SHU, signal:=od.do_4.bits[3]);

  (* Индикация ПС Фонарь   *)
  fb_AO_knopka_ind(str_SO := IM.SingleOutputs.AO_knopka_ind, signal:=od.do_4.bits[4]);

  (* Индикация АС Фонарь   *)
  fb_Pusk(str_SO := IM.SingleOutputs.Pusk_SHUP, signal:=od.do_4.bits[8]);

  (* Отключение МВ1 от КНА   *)
  fb_Stop_SHUP(str_SO := IM.SingleOutputs.Stop_SHUP, signal:=od.do_4.bits[9]);

  (* Отключение МВ1 от КНА   *)
  fb_NO_fonar(str_SO := IM.SingleOutputs.NO_fonar, signal:=od.do_3.bits[10]);

  (* Отключение МВ1 от КНА   *)
  fb_PC_fonar(str_SO := IM.SingleOutputs.PC_fonar, signal:=od.do_3.bits[9]);

  (* Отключение МВ1 от КНА   *)
  fb_AC_fonar(str_SO := IM.SingleOutputs.AC_fonar, signal:=od.do_3.bits[8]);

  (* Отключение МВ1 от КНА   *)
  fb_Kr1_smazka(str_SO := IM.SingleOutputs.Kr1_smazka, signal:=od.do_0.bits[14]);

  (* Отключение МВ1 от КНА   *)
  fb_Kr2_smazka(str_SO := IM.SingleOutputs.Kr2_smazka, signal:=od.do_0.bits[15]);

  (* Отключение МВ1 от КНА   *)
  fb_Kr4_open_from_alg(str_SO := IM.SingleOutputs.Kr4_open_from_alg, signal:=od.do_0.bits[8]);

  (* Отключение МВ1 от КНА   *)
  fb_Synch_rej_K1(str_SO := IM.SingleOutputs.Synch_rej_K1, signal:=od.do_3.bits[13]);

   (**************************************** Аналоговые и Дискретные параметры ***********************************)
END_FUNCTION_BLOCK

FUNCTION_BLOCK proc_DO_Init
  VAR_INPUT
    init : BOOL;
  END_VAR
  VAR
    stDO_Ini : fb_DO_Init;
    inits : UINT;
  END_VAR
  VAR_INPUT
    initiales : UINT;
  END_VAR
  VAR_EXTERNAL
    od : DOconfig;
  END_VAR

  (* Инициализация начало. Входные дискретные параметры *)

  inits := 0; (* Флаг необходимости инициализации структур-дескрипторов *)

  (* Модуль A1-15 *)
  stDO_Ini(data_Ini := true, imit:=FALSE, strDO := od.do_0);
  inits := inits + BOOL_TO_UINT(stDO_Ini.Init);

  (* Модуль A1-16 *)
  stDO_Ini(data_Ini := true, imit:=FALSE, strDO := od.do_1);
  inits := inits + BOOL_TO_UINT(stDO_Ini.Init);

  (* Модуль A1-17 *)
  stDO_Ini(data_Ini := true, imit:=FALSE, strDO := od.do_2);
  inits := inits + BOOL_TO_UINT(stDO_Ini.Init);

  (* Модуль A1-18 *)
  stDO_Ini(data_Ini := true, imit:=FALSE, strDO := od.do_3);
  inits := inits + BOOL_TO_UINT(stDO_Ini.Init);

  (* Модуль A1-19 *)
  stDO_Ini(data_Ini := true, imit:=FALSE, strDO := od.do_4);
  inits := inits + BOOL_TO_UINT(stDO_Ini.Init);

  (* Модуль A1-23 *)
  stDO_Ini(data_Ini := true, imit:=FALSE, strDO := od.gpio_out);
  inits := inits + BOOL_TO_UINT(stDO_Ini.Init);
  initiales := 0;

  IF init THEN initiales := inits; END_IF;
END_FUNCTION_BLOCK

FUNCTION_BLOCK OPC_algoritms_get
  VAR_EXTERNAL
    algoritms_autoNu : UINT;
    algoritms_AutoPns : UINT;
    algoritms_AutoAvom : UINT;
    algoritms_AutoTen : UINT;
    algoritms_AntiPompag : UINT;
    algoritms_testIm : UINT;
    algoritms_TestProtection : UINT;
    algoritms_Remont : UINT;
    algoritms_ppu : UINT;
    algoritms_puskOilSystem : UINT;
    algoritms_engineRun : UINT;
    algoritms_filling : UINT;
    algoritms_LineToRing : UINT;
    algoritms_RingToLine : UINT;
    algoritms_Apusk : UINT;
    algoritms_SemiAutoPusk : UINT;
    algoritms_no : UINT;
    algoritms_vibegPNS : UINT;
    algoritms_ao : UINT;
    algoritms_testPms : UINT;
    algoritms_testdPmg : UINT;
    algoritms_puskV : UINT;
    algoritms_puskK : UINT;
    algoritms_Pusk_F_faza1 : UINT;
    algoritms_Pusk_F_faza2 : UINT;
    algoritms_Pusk_TH_faza : UINT;
    algoritms_Prov_PMS_ALG : UINT;
    algoritms_Prov_opressovka_ALG : UINT;
    algoritms_Pusk_SEC_faza_chastotny : UINT;
    algoritms_Pusk_SEC_faza_reactor : UINT;
    algoritms : AlgoritmsConfig;
  END_VAR

  algoritms.autoNu.inCommand_ARM := UINT_TO_WORD(algoritms_autoNu);

  algoritms.AutoPns.inCommand_ARM := UINT_TO_WORD(algoritms_AutoPns);

  algoritms.AutoAvom.inCommand_ARM := UINT_TO_WORD(algoritms_AutoAvom);

  algoritms.AutoTen.inCommand_ARM := UINT_TO_WORD(algoritms_AutoTen);

  algoritms.AntiPompag.inCommand_ARM := UINT_TO_WORD(algoritms_AntiPompag);

  algoritms.testIm.inCommand_ARM := UINT_TO_WORD(algoritms_testIm);

  algoritms.TestProtection.inCommand_ARM := UINT_TO_WORD(algoritms_TestProtection);

  algoritms.Remont.inCommand_ARM := UINT_TO_WORD(algoritms_Remont);

  algoritms.ppu.inCommand_ARM := UINT_TO_WORD(algoritms_ppu);

  algoritms.puskOilSystem.inCommand_ARM := UINT_TO_WORD(algoritms_puskOilSystem);

  algoritms.engineRun.inCommand_ARM := UINT_TO_WORD(algoritms_engineRun);

  algoritms.filling.inCommand_ARM := UINT_TO_WORD(algoritms_filling);

  algoritms.LineToRing.inCommand_ARM := UINT_TO_WORD(algoritms_LineToRing);

  algoritms.RingToLine.inCommand_ARM := UINT_TO_WORD(algoritms_RingToLine);

  algoritms.Apusk.inCommand_ARM := UINT_TO_WORD(algoritms_Apusk);

  algoritms.SemiAutoPusk.inCommand_ARM := UINT_TO_WORD(algoritms_SemiAutoPusk);

  algoritms.no.inCommand_ARM := UINT_TO_WORD(algoritms_no);

  algoritms.vibegPNS.inCommand_ARM := UINT_TO_WORD(algoritms_vibegPNS);

  algoritms.ao.inCommand_ARM := UINT_TO_WORD(algoritms_ao);

  algoritms.testPms.inCommand_ARM := UINT_TO_WORD(algoritms_testPms);

  algoritms.testdPmg.inCommand_ARM := UINT_TO_WORD(algoritms_testdPmg);

  algoritms.puskV.inCommand_ARM := UINT_TO_WORD(algoritms_puskV);

  algoritms.puskK.inCommand_ARM := UINT_TO_WORD(algoritms_puskK);

  algoritms.Pusk_F_faza1.inCommand_ARM := UINT_TO_WORD(algoritms_Pusk_F_faza1);

  algoritms.Pusk_F_faza2.inCommand_ARM := UINT_TO_WORD(algoritms_Pusk_F_faza2);

  algoritms.Pusk_TH_faza.inCommand_ARM := UINT_TO_WORD(algoritms_Pusk_TH_faza);

  algoritms.Prov_PMS_ALG.inCommand_ARM := UINT_TO_WORD(algoritms_Prov_PMS_ALG);

  algoritms.Prov_opressovka_ALG.inCommand_ARM := UINT_TO_WORD(algoritms_Prov_opressovka_ALG);

  algoritms.Pusk_SEC_faza_chastotny.inCommand_ARM := UINT_TO_WORD(algoritms_Pusk_SEC_faza_chastotny);

  algoritms.Pusk_SEC_faza_reactor.inCommand_ARM := UINT_TO_WORD(algoritms_Pusk_SEC_faza_reactor);
END_FUNCTION_BLOCK

FUNCTION_BLOCK OPC_AI_SET
  VAR_EXTERNAL
    ai : aiConfig;
    AI_Tstali_statora_kanal_1_HL : LREAL;
    AI_Tstali_statora_kanal_1_LL : LREAL;
    AI_Tstali_statora_kanal_1_command : UINT;
    AI_Tstali_statora_kanal_1_newHL : LREAL;
    AI_Tstali_statora_kanal_1_newLL : LREAL;
    AI_Tstali_statora_kanal_1_status : UDINT;
    AI_Tstali_statora_kanal_1_value : LREAL;
    AI_Tstali_statora_kanal_1_HW : LREAL;
    AI_Tstali_statora_kanal_1_newHW : LREAL;
    AI_Tstali_statora_kanal_2_HL : LREAL;
    AI_Tstali_statora_kanal_2_LL : LREAL;
    AI_Tstali_statora_kanal_2_command : UINT;
    AI_Tstali_statora_kanal_2_newHL : LREAL;
    AI_Tstali_statora_kanal_2_newLL : LREAL;
    AI_Tstali_statora_kanal_2_status : UDINT;
    AI_Tstali_statora_kanal_2_value : LREAL;
    AI_Tstali_statora_kanal_2_HW : LREAL;
    AI_Tstali_statora_kanal_2_newHW : LREAL;
    AI_Tstali_statora_kanal_3_HL : LREAL;
    AI_Tstali_statora_kanal_3_LL : LREAL;
    AI_Tstali_statora_kanal_3_command : UINT;
    AI_Tstali_statora_kanal_3_newHL : LREAL;
    AI_Tstali_statora_kanal_3_newLL : LREAL;
    AI_Tstali_statora_kanal_3_status : UDINT;
    AI_Tstali_statora_kanal_3_value : LREAL;
    AI_Tstali_statora_kanal_3_HW : LREAL;
    AI_Tstali_statora_kanal_3_newHW : LREAL;
    AI_Tmedi_statora_kanal_1_HL : LREAL;
    AI_Tmedi_statora_kanal_1_LL : LREAL;
    AI_Tmedi_statora_kanal_1_command : UINT;
    AI_Tmedi_statora_kanal_1_newHL : LREAL;
    AI_Tmedi_statora_kanal_1_newLL : LREAL;
    AI_Tmedi_statora_kanal_1_status : UDINT;
    AI_Tmedi_statora_kanal_1_value : LREAL;
    AI_Tmedi_statora_kanal_1_HW : LREAL;
    AI_Tmedi_statora_kanal_1_newHW : LREAL;
    AI_Tmedi_statora_kanal_2_HL : LREAL;
    AI_Tmedi_statora_kanal_2_LL : LREAL;
    AI_Tmedi_statora_kanal_2_command : UINT;
    AI_Tmedi_statora_kanal_2_newHL : LREAL;
    AI_Tmedi_statora_kanal_2_newLL : LREAL;
    AI_Tmedi_statora_kanal_2_status : UDINT;
    AI_Tmedi_statora_kanal_2_value : LREAL;
    AI_Tmedi_statora_kanal_2_HW : LREAL;
    AI_Tmedi_statora_kanal_2_newHW : LREAL;
    AI_Tmedi_statora_kanal_3_HL : LREAL;
    AI_Tmedi_statora_kanal_3_LL : LREAL;
    AI_Tmedi_statora_kanal_3_command : UINT;
    AI_Tmedi_statora_kanal_3_newHL : LREAL;
    AI_Tmedi_statora_kanal_3_newLL : LREAL;
    AI_Tmedi_statora_kanal_3_status : UDINT;
    AI_Tmedi_statora_kanal_3_value : LREAL;
    AI_Tmedi_statora_kanal_3_HW : LREAL;
    AI_Tmedi_statora_kanal_3_newHW : LREAL;
    AI_Toporno_podshipnika_EDT_1_HL : LREAL;
    AI_Toporno_podshipnika_EDT_1_LL : LREAL;
    AI_Toporno_podshipnika_EDT_1_command : UINT;
    AI_Toporno_podshipnika_EDT_1_newHL : LREAL;
    AI_Toporno_podshipnika_EDT_1_newLL : LREAL;
    AI_Toporno_podshipnika_EDT_1_status : UDINT;
    AI_Toporno_podshipnika_EDT_1_value : LREAL;
    AI_Toporno_podshipnika_EDT_1_HW : LREAL;
    AI_Toporno_podshipnika_EDT_1_newHW : LREAL;
    AI_Toporno_podshipnika_EDT_1_HA : LREAL;
    AI_Toporno_podshipnika_EDT_1_newHA : LREAL;
    AI_Toy_podshipnika_EDT_2_HL : LREAL;
    AI_Toy_podshipnika_EDT_2_LL : LREAL;
    AI_Toy_podshipnika_EDT_2_command : UINT;
    AI_Toy_podshipnika_EDT_2_newHL : LREAL;
    AI_Toy_podshipnika_EDT_2_newLL : LREAL;
    AI_Toy_podshipnika_EDT_2_status : UDINT;
    AI_Toy_podshipnika_EDT_2_value : LREAL;
    AI_Toy_podshipnika_EDT_2_HW : LREAL;
    AI_Toy_podshipnika_EDT_2_newHW : LREAL;
    AI_Toy_podshipnika_EDT_2_HA : LREAL;
    AI_Toy_podshipnika_EDT_2_newHA : LREAL;
    AI_Toy_podshipnika_kol_EDT_3_HL : LREAL;
    AI_Toy_podshipnika_kol_EDT_3_LL : LREAL;
    AI_Toy_podshipnika_kol_EDT_3_command : UINT;
    AI_Toy_podshipnika_kol_EDT_3_newHL : LREAL;
    AI_Toy_podshipnika_kol_EDT_3_newLL : LREAL;
    AI_Toy_podshipnika_kol_EDT_3_status : UDINT;
    AI_Toy_podshipnika_kol_EDT_3_value : LREAL;
    AI_Toy_podshipnika_kol_EDT_3_HW : LREAL;
    AI_Toy_podshipnika_kol_EDT_3_newHW : LREAL;
    AI_Toy_podshipnika_kol_EDT_3_HA : LREAL;
    AI_Toy_podshipnika_kol_EDT_3_newHA : LREAL;
    AI_Toy_podshipnika_kol_EDT_4_HL : LREAL;
    AI_Toy_podshipnika_kol_EDT_4_LL : LREAL;
    AI_Toy_podshipnika_kol_EDT_4_command : UINT;
    AI_Toy_podshipnika_kol_EDT_4_newHL : LREAL;
    AI_Toy_podshipnika_kol_EDT_4_newLL : LREAL;
    AI_Toy_podshipnika_kol_EDT_4_status : UDINT;
    AI_Toy_podshipnika_kol_EDT_4_value : LREAL;
    AI_Toy_podshipnika_kol_EDT_4_HW : LREAL;
    AI_Toy_podshipnika_kol_EDT_4_newHW : LREAL;
    AI_Toy_podshipnika_kol_EDT_4_HA : LREAL;
    AI_Toy_podshipnika_kol_EDT_4_newHA : LREAL;
    AI_Toy_podshipnika_shest_red_EDT_5_HL : LREAL;
    AI_Toy_podshipnika_shest_red_EDT_5_LL : LREAL;
    AI_Toy_podshipnika_shest_red_EDT_5_command : UINT;
    AI_Toy_podshipnika_shest_red_EDT_5_newHL : LREAL;
    AI_Toy_podshipnika_shest_red_EDT_5_newLL : LREAL;
    AI_Toy_podshipnika_shest_red_EDT_5_status : UDINT;
    AI_Toy_podshipnika_shest_red_EDT_5_value : LREAL;
    AI_Toy_podshipnika_shest_red_EDT_5_HW : LREAL;
    AI_Toy_podshipnika_shest_red_EDT_5_newHW : LREAL;
    AI_Toy_podshipnika_shest_red_EDT_5_HA : LREAL;
    AI_Toy_podshipnika_shest_red_EDT_5_newHA : LREAL;
    AI_Ty_podshipnika_red_EDT_6_HL : LREAL;
    AI_Ty_podshipnika_red_EDT_6_LL : LREAL;
    AI_Ty_podshipnika_red_EDT_6_command : UINT;
    AI_Ty_podshipnika_red_EDT_6_newHL : LREAL;
    AI_Ty_podshipnika_red_EDT_6_newLL : LREAL;
    AI_Ty_podshipnika_red_EDT_6_status : UDINT;
    AI_Ty_podshipnika_red_EDT_6_value : LREAL;
    AI_Ty_podshipnika_red_EDT_6_HW : LREAL;
    AI_Ty_podshipnika_red_EDT_6_newHW : LREAL;
    AI_Ty_podshipnika_red_EDT_6_HA : LREAL;
    AI_Ty_podshipnika_red_EDT_6_newHA : LREAL;
    AI_Ty_podshipnika_nagnet_EDT_7_1_HL : LREAL;
    AI_Ty_podshipnika_nagnet_EDT_7_1_LL : LREAL;
    AI_Ty_podshipnika_nagnet_EDT_7_1_command : UINT;
    AI_Ty_podshipnika_nagnet_EDT_7_1_newHL : LREAL;
    AI_Ty_podshipnika_nagnet_EDT_7_1_newLL : LREAL;
    AI_Ty_podshipnika_nagnet_EDT_7_1_status : UDINT;
    AI_Ty_podshipnika_nagnet_EDT_7_1_value : LREAL;
    AI_Ty_podshipnika_nagnet_EDT_7_1_HW : LREAL;
    AI_Ty_podshipnika_nagnet_EDT_7_1_newHW : LREAL;
    AI_Ty_podshipnika_nagnet_EDT_7_1_HA : LREAL;
    AI_Ty_podshipnika_nagnet_EDT_7_1_newHA : LREAL;
    AI_Ty_podshipnika_nagnet_EDT_7_2_HL : LREAL;
    AI_Ty_podshipnika_nagnet_EDT_7_2_LL : LREAL;
    AI_Ty_podshipnika_nagnet_EDT_7_2_command : UINT;
    AI_Ty_podshipnika_nagnet_EDT_7_2_newHL : LREAL;
    AI_Ty_podshipnika_nagnet_EDT_7_2_newLL : LREAL;
    AI_Ty_podshipnika_nagnet_EDT_7_2_status : UDINT;
    AI_Ty_podshipnika_nagnet_EDT_7_2_value : LREAL;
    AI_Ty_podshipnika_nagnet_EDT_7_2_HW : LREAL;
    AI_Ty_podshipnika_nagnet_EDT_7_2_newHW : LREAL;
    AI_Ty_podshipnika_nagnet_EDT_7_2_HA : LREAL;
    AI_Ty_podshipnika_nagnet_EDT_7_2_newHA : LREAL;
    AI_Toy_podshipnika_svobod_konca_EDT_8_1_HL : LREAL;
    AI_Toy_podshipnika_svobod_konca_EDT_8_1_LL : LREAL;
    AI_Toy_podshipnika_svobod_konca_EDT_8_1_command : UINT;
    AI_Toy_podshipnika_svobod_konca_EDT_8_1_newHL : LREAL;
    AI_Toy_podshipnika_svobod_konca_EDT_8_1_newLL : LREAL;
    AI_Toy_podshipnika_svobod_konca_EDT_8_1_status : UDINT;
    AI_Toy_podshipnika_svobod_konca_EDT_8_1_value : LREAL;
    AI_Toy_podshipnika_svobod_konca_EDT_8_1_HW : LREAL;
    AI_Toy_podshipnika_svobod_konca_EDT_8_1_newHW : LREAL;
    AI_Toy_podshipnika_svobod_konca_EDT_8_1_HA : LREAL;
    AI_Toy_podshipnika_svobod_konca_EDT_8_1_newHA : LREAL;
    AI_Toy_podshipnika_svobod_konca_EDT_8_2_HL : LREAL;
    AI_Toy_podshipnika_svobod_konca_EDT_8_2_LL : LREAL;
    AI_Toy_podshipnika_svobod_konca_EDT_8_2_command : UINT;
    AI_Toy_podshipnika_svobod_konca_EDT_8_2_newHL : LREAL;
    AI_Toy_podshipnika_svobod_konca_EDT_8_2_newLL : LREAL;
    AI_Toy_podshipnika_svobod_konca_EDT_8_2_status : UDINT;
    AI_Toy_podshipnika_svobod_konca_EDT_8_2_value : LREAL;
    AI_Toy_podshipnika_svobod_konca_EDT_8_2_HW : LREAL;
    AI_Toy_podshipnika_svobod_konca_EDT_8_2_newHW : LREAL;
    AI_Toy_podshipnika_svobod_konca_EDT_8_2_HA : LREAL;
    AI_Toy_podshipnika_svobod_konca_EDT_8_2_newHA : LREAL;
    AI_Toy_podshipnika_rab_kol_EDT_9_1_HL : LREAL;
    AI_Toy_podshipnika_rab_kol_EDT_9_1_LL : LREAL;
    AI_Toy_podshipnika_rab_kol_EDT_9_1_command : UINT;
    AI_Toy_podshipnika_rab_kol_EDT_9_1_newHL : LREAL;
    AI_Toy_podshipnika_rab_kol_EDT_9_1_newLL : LREAL;
    AI_Toy_podshipnika_rab_kol_EDT_9_1_status : UDINT;
    AI_Toy_podshipnika_rab_kol_EDT_9_1_value : LREAL;
    AI_Toy_podshipnika_rab_kol_EDT_9_1_HW : LREAL;
    AI_Toy_podshipnika_rab_kol_EDT_9_1_newHW : LREAL;
    AI_Toy_podshipnika_rab_kol_EDT_9_1_HA : LREAL;
    AI_Toy_podshipnika_rab_kol_EDT_9_1_newHA : LREAL;
    AI_Toy_podshipnika_rab_kol_EDT_9_2_HL : LREAL;
    AI_Toy_podshipnika_rab_kol_EDT_9_2_LL : LREAL;
    AI_Toy_podshipnika_rab_kol_EDT_9_2_command : UINT;
    AI_Toy_podshipnika_rab_kol_EDT_9_2_newHL : LREAL;
    AI_Toy_podshipnika_rab_kol_EDT_9_2_newLL : LREAL;
    AI_Toy_podshipnika_rab_kol_EDT_9_2_status : UDINT;
    AI_Toy_podshipnika_rab_kol_EDT_9_2_value : LREAL;
    AI_Toy_podshipnika_rab_kol_EDT_9_2_HW : LREAL;
    AI_Toy_podshipnika_rab_kol_EDT_9_2_newHW : LREAL;
    AI_Toy_podshipnika_rab_kol_EDT_9_2_HA : LREAL;
    AI_Toy_podshipnika_rab_kol_EDT_9_2_newHA : LREAL;
    AI_Toy_podshipnika_nerab_kol_EDT_10_1_HL : LREAL;
    AI_Toy_podshipnika_nerab_kol_EDT_10_1_LL : LREAL;
    AI_Toy_podshipnika_nerab_kol_EDT_10_1_command : UINT;
    AI_Toy_podshipnika_nerab_kol_EDT_10_1_newHL : LREAL;
    AI_Toy_podshipnika_nerab_kol_EDT_10_1_newLL : LREAL;
    AI_Toy_podshipnika_nerab_kol_EDT_10_1_status : UDINT;
    AI_Toy_podshipnika_nerab_kol_EDT_10_1_value : LREAL;
    AI_Toy_podshipnika_nerab_kol_EDT_10_1_HW : LREAL;
    AI_Toy_podshipnika_nerab_kol_EDT_10_1_newHW : LREAL;
    AI_Toy_podshipnika_nerab_kol_EDT_10_1_HA : LREAL;
    AI_Toy_podshipnika_nerab_kol_EDT_10_1_newHA : LREAL;
    AI_Toy_podshipnika_nerab_kol_EDT_10_2_HL : LREAL;
    AI_Toy_podshipnika_nerab_kol_EDT_10_2_LL : LREAL;
    AI_Toy_podshipnika_nerab_kol_EDT_10_2_command : UINT;
    AI_Toy_podshipnika_nerab_kol_EDT_10_2_newHL : LREAL;
    AI_Toy_podshipnika_nerab_kol_EDT_10_2_newLL : LREAL;
    AI_Toy_podshipnika_nerab_kol_EDT_10_2_status : UDINT;
    AI_Toy_podshipnika_nerab_kol_EDT_10_2_value : LREAL;
    AI_Toy_podshipnika_nerab_kol_EDT_10_2_HW : LREAL;
    AI_Toy_podshipnika_nerab_kol_EDT_10_2_newHW : LREAL;
    AI_Toy_podshipnika_nerab_kol_EDT_10_2_HA : LREAL;
    AI_Toy_podshipnika_nerab_kol_EDT_10_2_newHA : LREAL;
    AI_Tholodnogo_vozduha_ED_kanal_1_HL : LREAL;
    AI_Tholodnogo_vozduha_ED_kanal_1_LL : LREAL;
    AI_Tholodnogo_vozduha_ED_kanal_1_command : UINT;
    AI_Tholodnogo_vozduha_ED_kanal_1_newHL : LREAL;
    AI_Tholodnogo_vozduha_ED_kanal_1_newLL : LREAL;
    AI_Tholodnogo_vozduha_ED_kanal_1_status : UDINT;
    AI_Tholodnogo_vozduha_ED_kanal_1_value : LREAL;
    AI_Tholodnogo_vozduha_ED_kanal_1_HW : LREAL;
    AI_Tholodnogo_vozduha_ED_kanal_1_newHW : LREAL;
    AI_Tholodnogo_vozduha_ED_kanal_2_HL : LREAL;
    AI_Tholodnogo_vozduha_ED_kanal_2_LL : LREAL;
    AI_Tholodnogo_vozduha_ED_kanal_2_command : UINT;
    AI_Tholodnogo_vozduha_ED_kanal_2_newHL : LREAL;
    AI_Tholodnogo_vozduha_ED_kanal_2_newLL : LREAL;
    AI_Tholodnogo_vozduha_ED_kanal_2_status : UDINT;
    AI_Tholodnogo_vozduha_ED_kanal_2_value : LREAL;
    AI_Tholodnogo_vozduha_ED_kanal_2_HW : LREAL;
    AI_Tholodnogo_vozduha_ED_kanal_2_newHW : LREAL;
    AI_Tgorjachego_vozduha_ED_kanal_1_HL : LREAL;
    AI_Tgorjachego_vozduha_ED_kanal_1_LL : LREAL;
    AI_Tgorjachego_vozduha_ED_kanal_1_command : UINT;
    AI_Tgorjachego_vozduha_ED_kanal_1_newHL : LREAL;
    AI_Tgorjachego_vozduha_ED_kanal_1_newLL : LREAL;
    AI_Tgorjachego_vozduha_ED_kanal_1_status : UDINT;
    AI_Tgorjachego_vozduha_ED_kanal_1_value : LREAL;
    AI_Tgorjachego_vozduha_ED_kanal_1_HW : LREAL;
    AI_Tgorjachego_vozduha_ED_kanal_1_newHW : LREAL;
    AI_Tgorjachego_vozduha_ED_kanal_2_HL : LREAL;
    AI_Tgorjachego_vozduha_ED_kanal_2_LL : LREAL;
    AI_Tgorjachego_vozduha_ED_kanal_2_command : UINT;
    AI_Tgorjachego_vozduha_ED_kanal_2_newHL : LREAL;
    AI_Tgorjachego_vozduha_ED_kanal_2_newLL : LREAL;
    AI_Tgorjachego_vozduha_ED_kanal_2_status : UDINT;
    AI_Tgorjachego_vozduha_ED_kanal_2_value : LREAL;
    AI_Tgorjachego_vozduha_ED_kanal_2_HW : LREAL;
    AI_Tgorjachego_vozduha_ED_kanal_2_newHW : LREAL;
    AI_Tnarujnogo_vozduha_HL : LREAL;
    AI_Tnarujnogo_vozduha_LL : LREAL;
    AI_Tnarujnogo_vozduha_command : UINT;
    AI_Tnarujnogo_vozduha_newHL : LREAL;
    AI_Tnarujnogo_vozduha_newLL : LREAL;
    AI_Tnarujnogo_vozduha_status : UDINT;
    AI_Tnarujnogo_vozduha_value : LREAL;
    AI_Tnarujnogo_vozduha_HW : LREAL;
    AI_Tnarujnogo_vozduha_newHW : LREAL;
    AI_Tgaza_na_vhode_H_HL : LREAL;
    AI_Tgaza_na_vhode_H_LL : LREAL;
    AI_Tgaza_na_vhode_H_command : UINT;
    AI_Tgaza_na_vhode_H_newHL : LREAL;
    AI_Tgaza_na_vhode_H_newLL : LREAL;
    AI_Tgaza_na_vhode_H_status : UDINT;
    AI_Tgaza_na_vhode_H_value : LREAL;
    AI_Tgaza_na_vhode_H_HW : LREAL;
    AI_Tgaza_na_vhode_H_newHW : LREAL;
    AI_Tgaza_na_vyhode_H_HL : LREAL;
    AI_Tgaza_na_vyhode_H_LL : LREAL;
    AI_Tgaza_na_vyhode_H_command : UINT;
    AI_Tgaza_na_vyhode_H_newHL : LREAL;
    AI_Tgaza_na_vyhode_H_newLL : LREAL;
    AI_Tgaza_na_vyhode_H_status : UDINT;
    AI_Tgaza_na_vyhode_H_value : LREAL;
    AI_Tgaza_na_vyhode_H_HW : LREAL;
    AI_Tgaza_na_vyhode_H_newHW : LREAL;
    AI_Tgaza_na_vyhode_H_HA : LREAL;
    AI_Tgaza_na_vyhode_H_newHA : LREAL;
    AI_Tmasla_do_AVOM_HL : LREAL;
    AI_Tmasla_do_AVOM_LL : LREAL;
    AI_Tmasla_do_AVOM_command : UINT;
    AI_Tmasla_do_AVOM_newHL : LREAL;
    AI_Tmasla_do_AVOM_newLL : LREAL;
    AI_Tmasla_do_AVOM_status : UDINT;
    AI_Tmasla_do_AVOM_value : LREAL;
    AI_Tmasla_do_AVOM_HW : LREAL;
    AI_Tmasla_do_AVOM_newHW : LREAL;
    AI_Tmasla_posle_AVOM_HL : LREAL;
    AI_Tmasla_posle_AVOM_LL : LREAL;
    AI_Tmasla_posle_AVOM_command : UINT;
    AI_Tmasla_posle_AVOM_newHL : LREAL;
    AI_Tmasla_posle_AVOM_newLL : LREAL;
    AI_Tmasla_posle_AVOM_status : UDINT;
    AI_Tmasla_posle_AVOM_value : LREAL;
    AI_Tmasla_posle_AVOM_HW : LREAL;
    AI_Tmasla_posle_AVOM_newHW : LREAL;
    AI_Tmasla_MB_HL : LREAL;
    AI_Tmasla_MB_LL : LREAL;
    AI_Tmasla_MB_command : UINT;
    AI_Tmasla_MB_newHL : LREAL;
    AI_Tmasla_MB_newLL : LREAL;
    AI_Tmasla_MB_status : UDINT;
    AI_Tmasla_MB_value : LREAL;
    AI_Tmasla_MB_HW : LREAL;
    AI_Tmasla_MB_newHW : LREAL;
    AI_Tmasla_MB_TEN_HL : LREAL;
    AI_Tmasla_MB_TEN_LL : LREAL;
    AI_Tmasla_MB_TEN_command : UINT;
    AI_Tmasla_MB_TEN_newHL : LREAL;
    AI_Tmasla_MB_TEN_newLL : LREAL;
    AI_Tmasla_MB_TEN_status : UDINT;
    AI_Tmasla_MB_TEN_value : LREAL;
    AI_Tmasla_MB_TEN_HW : LREAL;
    AI_Tmasla_MB_TEN_newHW : LREAL;
    AI_Tshu_HL : LREAL;
    AI_Tshu_LL : LREAL;
    AI_Tshu_command : UINT;
    AI_Tshu_newHL : LREAL;
    AI_Tshu_newLL : LREAL;
    AI_Tshu_status : UDINT;
    AI_Tshu_value : LREAL;
    AI_Pmaslo_sm_nizkoe_HL : LREAL;
    AI_Pmaslo_sm_nizkoe_LL : LREAL;
    AI_Pmaslo_sm_nizkoe_command : UINT;
    AI_Pmaslo_sm_nizkoe_newHL : LREAL;
    AI_Pmaslo_sm_nizkoe_newLL : LREAL;
    AI_Pmaslo_sm_nizkoe_status : UDINT;
    AI_Pmaslo_sm_nizkoe_value : LREAL;
    AI_Pmaslo_sm_nizkoe_LW : LREAL;
    AI_Pmaslo_sm_nizkoe_newLW : LREAL;
    AI_Pmaslo_sm_nizkoe_LA : LREAL;
    AI_Pmaslo_sm_nizkoe_newLA : LREAL;
    AI_Pmaslo_sm_vysokoe_HL : LREAL;
    AI_Pmaslo_sm_vysokoe_LL : LREAL;
    AI_Pmaslo_sm_vysokoe_command : UINT;
    AI_Pmaslo_sm_vysokoe_newHL : LREAL;
    AI_Pmaslo_sm_vysokoe_newLL : LREAL;
    AI_Pmaslo_sm_vysokoe_status : UDINT;
    AI_Pmaslo_sm_vysokoe_value : LREAL;
    AI_Pmaslo_sm_vysokoe_LW : LREAL;
    AI_Pmaslo_sm_vysokoe_newLW : LREAL;
    AI_Pmaslo_sm_vysokoe_LA : LREAL;
    AI_Pmaslo_sm_vysokoe_newLA : LREAL;
    AI_Pmasla_posle_GNS_HL : LREAL;
    AI_Pmasla_posle_GNS_LL : LREAL;
    AI_Pmasla_posle_GNS_command : UINT;
    AI_Pmasla_posle_GNS_newHL : LREAL;
    AI_Pmasla_posle_GNS_newLL : LREAL;
    AI_Pmasla_posle_GNS_status : UDINT;
    AI_Pmasla_posle_GNS_value : LREAL;
    AI_Pmasla_posle_GNS_HW : LREAL;
    AI_Pmasla_posle_GNS_newHW : LREAL;
    AI_Pmasla_posle_GNS_LW : LREAL;
    AI_Pmasla_posle_GNS_newLW : LREAL;
    AI_Pmasla_posle_NU_HL : LREAL;
    AI_Pmasla_posle_NU_LL : LREAL;
    AI_Pmasla_posle_NU_command : UINT;
    AI_Pmasla_posle_NU_newHL : LREAL;
    AI_Pmasla_posle_NU_newLL : LREAL;
    AI_Pmasla_posle_NU_status : UDINT;
    AI_Pmasla_posle_NU_value : LREAL;
    AI_Pmasla_posle_NU_LW : LREAL;
    AI_Pmasla_posle_NU_newLW : LREAL;
    AI_Pgaza_na_vhode_nagnetatelia_HL : LREAL;
    AI_Pgaza_na_vhode_nagnetatelia_LL : LREAL;
    AI_Pgaza_na_vhode_nagnetatelia_command : UINT;
    AI_Pgaza_na_vhode_nagnetatelia_newHL : LREAL;
    AI_Pgaza_na_vhode_nagnetatelia_newLL : LREAL;
    AI_Pgaza_na_vhode_nagnetatelia_status : UDINT;
    AI_Pgaza_na_vhode_nagnetatelia_value : LREAL;
    AI_Pgaza_na_vhode_nagnetatelia_LW : LREAL;
    AI_Pgaza_na_vhode_nagnetatelia_newLW : LREAL;
    AI_Pgaza_na_vyhode_nagnetatelia_HL : LREAL;
    AI_Pgaza_na_vyhode_nagnetatelia_LL : LREAL;
    AI_Pgaza_na_vyhode_nagnetatelia_command : UINT;
    AI_Pgaza_na_vyhode_nagnetatelia_newHL : LREAL;
    AI_Pgaza_na_vyhode_nagnetatelia_newLL : LREAL;
    AI_Pgaza_na_vyhode_nagnetatelia_status : UDINT;
    AI_Pgaza_na_vyhode_nagnetatelia_value : LREAL;
    AI_Pgaza_na_vyhode_nagnetatelia_LW : LREAL;
    AI_Pgaza_na_vyhode_nagnetatelia_newLW : LREAL;
    AI_Pgaza_na_vyhode_nagnetatelia_HA : LREAL;
    AI_Pgaza_na_vyhode_nagnetatelia_newHA : LREAL;
    AI_Pimpuls_gaz_HL : LREAL;
    AI_Pimpuls_gaz_LL : LREAL;
    AI_Pimpuls_gaz_command : UINT;
    AI_Pimpuls_gaz_newHL : LREAL;
    AI_Pimpuls_gaz_newLL : LREAL;
    AI_Pimpuls_gaz_status : UDINT;
    AI_Pimpuls_gaz_value : LREAL;
    AI_Pimpuls_gaz_LW : LREAL;
    AI_Pimpuls_gaz_newLW : LREAL;
    AI_dPgaza_na_maslo_filtre_HL : LREAL;
    AI_dPgaza_na_maslo_filtre_LL : LREAL;
    AI_dPgaza_na_maslo_filtre_command : UINT;
    AI_dPgaza_na_maslo_filtre_newHL : LREAL;
    AI_dPgaza_na_maslo_filtre_newLL : LREAL;
    AI_dPgaza_na_maslo_filtre_status : UDINT;
    AI_dPgaza_na_maslo_filtre_value : LREAL;
    AI_dPgaza_na_maslo_filtre_HW : LREAL;
    AI_dPgaza_na_maslo_filtre_newHW : LREAL;
    AI_dPgaza_na_konfuzore_HL : LREAL;
    AI_dPgaza_na_konfuzore_LL : LREAL;
    AI_dPgaza_na_konfuzore_command : UINT;
    AI_dPgaza_na_konfuzore_newHL : LREAL;
    AI_dPgaza_na_konfuzore_newLL : LREAL;
    AI_dPgaza_na_konfuzore_status : UDINT;
    AI_dPgaza_na_konfuzore_value : LREAL;
    AI_dPgaza_na_konfuzore_LW : LREAL;
    AI_dPgaza_na_konfuzore_newLW : LREAL;
    AI_dPmaslo_gaz_HL : LREAL;
    AI_dPmaslo_gaz_LL : LREAL;
    AI_dPmaslo_gaz_command : UINT;
    AI_dPmaslo_gaz_newHL : LREAL;
    AI_dPmaslo_gaz_newLL : LREAL;
    AI_dPmaslo_gaz_status : UDINT;
    AI_dPmaslo_gaz_value : LREAL;
    AI_dPmaslo_gaz_LW : LREAL;
    AI_dPmaslo_gaz_newLW : LREAL;
    AI_dPmaslo_gaz_LA : LREAL;
    AI_dPmaslo_gaz_newLA : LREAL;
    AI_Os_sdvig_nagnetatelja_plus_HL : LREAL;
    AI_Os_sdvig_nagnetatelja_plus_LL : LREAL;
    AI_Os_sdvig_nagnetatelja_plus_command : UINT;
    AI_Os_sdvig_nagnetatelja_plus_newHL : LREAL;
    AI_Os_sdvig_nagnetatelja_plus_newLL : LREAL;
    AI_Os_sdvig_nagnetatelja_plus_status : UDINT;
    AI_Os_sdvig_nagnetatelja_plus_value : LREAL;
    AI_Os_sdvig_nagnetatelja_plus_HW : LREAL;
    AI_Os_sdvig_nagnetatelja_plus_newHW : LREAL;
    AI_Os_sdvig_nagnetatelja_plus_HA : LREAL;
    AI_Os_sdvig_nagnetatelja_plus_newHA : LREAL;
    AI_Os_sdvig_nagnetatelja_minus_HL : LREAL;
    AI_Os_sdvig_nagnetatelja_minus_LL : LREAL;
    AI_Os_sdvig_nagnetatelja_minus_command : UINT;
    AI_Os_sdvig_nagnetatelja_minus_newHL : LREAL;
    AI_Os_sdvig_nagnetatelja_minus_newLL : LREAL;
    AI_Os_sdvig_nagnetatelja_minus_status : UDINT;
    AI_Os_sdvig_nagnetatelja_minus_value : LREAL;
    AI_Os_sdvig_nagnetatelja_minus_LW : LREAL;
    AI_Os_sdvig_nagnetatelja_minus_newLW : LREAL;
    AI_Os_sdvig_nagnetatelja_minus_LA : LREAL;
    AI_Os_sdvig_nagnetatelja_minus_newLA : LREAL;
    AI_Yroven_masla_MB_HL : LREAL;
    AI_Yroven_masla_MB_LL : LREAL;
    AI_Yroven_masla_MB_command : UINT;
    AI_Yroven_masla_MB_newHL : LREAL;
    AI_Yroven_masla_MB_newLL : LREAL;
    AI_Yroven_masla_MB_status : UDINT;
    AI_Yroven_masla_MB_value : LREAL;
    AI_Yroven_masla_MB_LW : LREAL;
    AI_Yroven_masla_MB_newLW : LREAL;
    AI_Kontrol_per_220V_HL : LREAL;
    AI_Kontrol_per_220V_LL : LREAL;
    AI_Kontrol_per_220V_command : UINT;
    AI_Kontrol_per_220V_newHL : LREAL;
    AI_Kontrol_per_220V_newLL : LREAL;
    AI_Kontrol_per_220V_status : UDINT;
    AI_Kontrol_per_220V_value : LREAL;
    AI_Kontrol_per_220V_HW : LREAL;
    AI_Kontrol_per_220V_newHW : LREAL;
    AI_Kontrol_per_220V_LW : LREAL;
    AI_Kontrol_per_220V_newLW : LREAL;
    AI_Kontrol_post_220V_HL : LREAL;
    AI_Kontrol_post_220V_LL : LREAL;
    AI_Kontrol_post_220V_command : UINT;
    AI_Kontrol_post_220V_newHL : LREAL;
    AI_Kontrol_post_220V_newLL : LREAL;
    AI_Kontrol_post_220V_status : UDINT;
    AI_Kontrol_post_220V_value : LREAL;
    AI_Kontrol_post_220V_HW : LREAL;
    AI_Kontrol_post_220V_newHW : LREAL;
    AI_Kontrol_post_220V_LW : LREAL;
    AI_Kontrol_post_220V_newLW : LREAL;
    AI_Tok_statora_HL : LREAL;
    AI_Tok_statora_LL : LREAL;
    AI_Tok_statora_command : UINT;
    AI_Tok_statora_newHL : LREAL;
    AI_Tok_statora_newLL : LREAL;
    AI_Tok_statora_status : UDINT;
    AI_Tok_statora_value : LREAL;
    AI_Tok_statora_LW : LREAL;
    AI_Tok_statora_newLW : LREAL;
    AI_Vibro_skorost_OPED_T1_HL : LREAL;
    AI_Vibro_skorost_OPED_T1_LL : LREAL;
    AI_Vibro_skorost_OPED_T1_command : UINT;
    AI_Vibro_skorost_OPED_T1_newHL : LREAL;
    AI_Vibro_skorost_OPED_T1_newLL : LREAL;
    AI_Vibro_skorost_OPED_T1_status : UDINT;
    AI_Vibro_skorost_OPED_T1_value : LREAL;
    AI_Vibro_skorost_OPED_T1_HW : LREAL;
    AI_Vibro_skorost_OPED_T1_newHW : LREAL;
    AI_Vibro_skorost_OPED_T1_HA : LREAL;
    AI_Vibro_skorost_OPED_T1_newHA : LREAL;
    AI_Vibro_skorost_OYPED_T2_HL : LREAL;
    AI_Vibro_skorost_OYPED_T2_LL : LREAL;
    AI_Vibro_skorost_OYPED_T2_command : UINT;
    AI_Vibro_skorost_OYPED_T2_newHL : LREAL;
    AI_Vibro_skorost_OYPED_T2_newLL : LREAL;
    AI_Vibro_skorost_OYPED_T2_status : UDINT;
    AI_Vibro_skorost_OYPED_T2_value : LREAL;
    AI_Vibro_skorost_OYPED_T2_HW : LREAL;
    AI_Vibro_skorost_OYPED_T2_newHW : LREAL;
    AI_Vibro_skorost_OYPED_T2_HA : LREAL;
    AI_Vibro_skorost_OYPED_T2_newHA : LREAL;
    AI_Vibro_skorost_OYP_kolesa_ED_T3_HL : LREAL;
    AI_Vibro_skorost_OYP_kolesa_ED_T3_LL : LREAL;
    AI_Vibro_skorost_OYP_kolesa_ED_T3_command : UINT;
    AI_Vibro_skorost_OYP_kolesa_ED_T3_newHL : LREAL;
    AI_Vibro_skorost_OYP_kolesa_ED_T3_newLL : LREAL;
    AI_Vibro_skorost_OYP_kolesa_ED_T3_status : UDINT;
    AI_Vibro_skorost_OYP_kolesa_ED_T3_value : LREAL;
    AI_Vibro_skorost_OYP_kolesa_ED_T3_HW : LREAL;
    AI_Vibro_skorost_OYP_kolesa_ED_T3_newHW : LREAL;
    AI_Vibro_skorost_OYP_kolesa_ED_T3_HA : LREAL;
    AI_Vibro_skorost_OYP_kolesa_ED_T3_newHA : LREAL;
    AI_Vibro_skorost_OP_kolesa_RH_T4_HL : LREAL;
    AI_Vibro_skorost_OP_kolesa_RH_T4_LL : LREAL;
    AI_Vibro_skorost_OP_kolesa_RH_T4_command : UINT;
    AI_Vibro_skorost_OP_kolesa_RH_T4_newHL : LREAL;
    AI_Vibro_skorost_OP_kolesa_RH_T4_newLL : LREAL;
    AI_Vibro_skorost_OP_kolesa_RH_T4_status : UDINT;
    AI_Vibro_skorost_OP_kolesa_RH_T4_value : LREAL;
    AI_Vibro_skorost_OP_kolesa_RH_T4_HW : LREAL;
    AI_Vibro_skorost_OP_kolesa_RH_T4_newHW : LREAL;
    AI_Vibro_skorost_OP_kolesa_RH_T4_HA : LREAL;
    AI_Vibro_skorost_OP_kolesa_RH_T4_newHA : LREAL;
    AI_Vibro_skorost_OP_shesterni_RED_T5_HL : LREAL;
    AI_Vibro_skorost_OP_shesterni_RED_T5_LL : LREAL;
    AI_Vibro_skorost_OP_shesterni_RED_T5_command : UINT;
    AI_Vibro_skorost_OP_shesterni_RED_T5_newHL : LREAL;
    AI_Vibro_skorost_OP_shesterni_RED_T5_newLL : LREAL;
    AI_Vibro_skorost_OP_shesterni_RED_T5_status : UDINT;
    AI_Vibro_skorost_OP_shesterni_RED_T5_value : LREAL;
    AI_Vibro_skorost_OP_shesterni_RED_T5_HW : LREAL;
    AI_Vibro_skorost_OP_shesterni_RED_T5_newHW : LREAL;
    AI_Vibro_skorost_OP_shesterni_RED_T5_HA : LREAL;
    AI_Vibro_skorost_OP_shesterni_RED_T5_newHA : LREAL;
    AI_Vibro_skorost_OP_shesterni_RED_T6_HL : LREAL;
    AI_Vibro_skorost_OP_shesterni_RED_T6_LL : LREAL;
    AI_Vibro_skorost_OP_shesterni_RED_T6_command : UINT;
    AI_Vibro_skorost_OP_shesterni_RED_T6_newHL : LREAL;
    AI_Vibro_skorost_OP_shesterni_RED_T6_newLL : LREAL;
    AI_Vibro_skorost_OP_shesterni_RED_T6_status : UDINT;
    AI_Vibro_skorost_OP_shesterni_RED_T6_value : LREAL;
    AI_Vibro_skorost_OP_shesterni_RED_T6_HW : LREAL;
    AI_Vibro_skorost_OP_shesterni_RED_T6_newHW : LREAL;
    AI_Vibro_skorost_OP_shesterni_RED_T6_HA : LREAL;
    AI_Vibro_skorost_OP_shesterni_RED_T6_newHA : LREAL;
  END_VAR

  AI_Tstali_statora_kanal_1_HL := ai.Tstali_statora_kanal_1.HL;
  AI_Tstali_statora_kanal_1_LL := ai.Tstali_statora_kanal_1.LL;
  AI_Tstali_statora_kanal_1_status := DWORD_TO_UDINT(ai.Tstali_statora_kanal_1.status);
  AI_Tstali_statora_kanal_1_value := ai.Tstali_statora_kanal_1.value;
  AI_Tstali_statora_kanal_1_HW := ai.Tstali_statora_kanal_1.HW;

  AI_Tstali_statora_kanal_2_HL := ai.Tstali_statora_kanal_2.HL;
  AI_Tstali_statora_kanal_2_LL := ai.Tstali_statora_kanal_2.LL;
  AI_Tstali_statora_kanal_2_status := DWORD_TO_UDINT(ai.Tstali_statora_kanal_2.status);
  AI_Tstali_statora_kanal_2_value := ai.Tstali_statora_kanal_2.value;
  AI_Tstali_statora_kanal_2_HW := ai.Tstali_statora_kanal_2.HW;

  AI_Tstali_statora_kanal_3_HL := ai.Tstali_statora_kanal_3.HL;
  AI_Tstali_statora_kanal_3_LL := ai.Tstali_statora_kanal_3.LL;
  AI_Tstali_statora_kanal_3_status := DWORD_TO_UDINT(ai.Tstali_statora_kanal_3.status);
  AI_Tstali_statora_kanal_3_value := ai.Tstali_statora_kanal_3.value;
  AI_Tstali_statora_kanal_3_HW := ai.Tstali_statora_kanal_3.HW;

  AI_Tmedi_statora_kanal_1_HL := ai.Tmedi_statora_kanal_1.HL;
  AI_Tmedi_statora_kanal_1_LL := ai.Tmedi_statora_kanal_1.LL;
  AI_Tmedi_statora_kanal_1_status := DWORD_TO_UDINT(ai.Tmedi_statora_kanal_1.status);
  AI_Tmedi_statora_kanal_1_value := ai.Tmedi_statora_kanal_1.value;
  AI_Tmedi_statora_kanal_1_HW := ai.Tmedi_statora_kanal_1.HW;

  AI_Tmedi_statora_kanal_2_HL := ai.Tmedi_statora_kanal_2.HL;
  AI_Tmedi_statora_kanal_2_LL := ai.Tmedi_statora_kanal_2.LL;
  AI_Tmedi_statora_kanal_2_status := DWORD_TO_UDINT(ai.Tmedi_statora_kanal_2.status);
  AI_Tmedi_statora_kanal_2_value := ai.Tmedi_statora_kanal_2.value;
  AI_Tmedi_statora_kanal_2_HW := ai.Tmedi_statora_kanal_2.HW;

  AI_Tmedi_statora_kanal_3_HL := ai.Tmedi_statora_kanal_3.HL;
  AI_Tmedi_statora_kanal_3_LL := ai.Tmedi_statora_kanal_3.LL;
  AI_Tmedi_statora_kanal_3_status := DWORD_TO_UDINT(ai.Tmedi_statora_kanal_3.status);
  AI_Tmedi_statora_kanal_3_value := ai.Tmedi_statora_kanal_3.value;
  AI_Tmedi_statora_kanal_3_HW := ai.Tmedi_statora_kanal_3.HW;

  AI_Toporno_podshipnika_EDT_1_HL := ai.Toporno_podshipnika_EDT_1.HL;
  AI_Toporno_podshipnika_EDT_1_LL := ai.Toporno_podshipnika_EDT_1.LL;
  AI_Toporno_podshipnika_EDT_1_status := DWORD_TO_UDINT(ai.Toporno_podshipnika_EDT_1.status);
  AI_Toporno_podshipnika_EDT_1_value := ai.Toporno_podshipnika_EDT_1.value;
  AI_Toporno_podshipnika_EDT_1_HW := ai.Toporno_podshipnika_EDT_1.HW;
  AI_Toporno_podshipnika_EDT_1_HA := ai.Toporno_podshipnika_EDT_1.HA;

  AI_Toy_podshipnika_EDT_2_HL := ai.Toy_podshipnika_EDT_2.HL;
  AI_Toy_podshipnika_EDT_2_LL := ai.Toy_podshipnika_EDT_2.LL;
  AI_Toy_podshipnika_EDT_2_status := DWORD_TO_UDINT(ai.Toy_podshipnika_EDT_2.status);
  AI_Toy_podshipnika_EDT_2_value := ai.Toy_podshipnika_EDT_2.value;
  AI_Toy_podshipnika_EDT_2_HW := ai.Toy_podshipnika_EDT_2.HW;
  AI_Toy_podshipnika_EDT_2_HA := ai.Toy_podshipnika_EDT_2.HA;

  AI_Toy_podshipnika_kol_EDT_3_HL := ai.Toy_podshipnika_kol_EDT_3.HL;
  AI_Toy_podshipnika_kol_EDT_3_LL := ai.Toy_podshipnika_kol_EDT_3.LL;
  AI_Toy_podshipnika_kol_EDT_3_status := DWORD_TO_UDINT(ai.Toy_podshipnika_kol_EDT_3.status);
  AI_Toy_podshipnika_kol_EDT_3_value := ai.Toy_podshipnika_kol_EDT_3.value;
  AI_Toy_podshipnika_kol_EDT_3_HW := ai.Toy_podshipnika_kol_EDT_3.HW;
  AI_Toy_podshipnika_kol_EDT_3_HA := ai.Toy_podshipnika_kol_EDT_3.HA;

  AI_Toy_podshipnika_kol_EDT_4_HL := ai.Toy_podshipnika_kol_EDT_4.HL;
  AI_Toy_podshipnika_kol_EDT_4_LL := ai.Toy_podshipnika_kol_EDT_4.LL;
  AI_Toy_podshipnika_kol_EDT_4_status := DWORD_TO_UDINT(ai.Toy_podshipnika_kol_EDT_4.status);
  AI_Toy_podshipnika_kol_EDT_4_value := ai.Toy_podshipnika_kol_EDT_4.value;
  AI_Toy_podshipnika_kol_EDT_4_HW := ai.Toy_podshipnika_kol_EDT_4.HW;
  AI_Toy_podshipnika_kol_EDT_4_HA := ai.Toy_podshipnika_kol_EDT_4.HA;

  AI_Toy_podshipnika_shest_red_EDT_5_HL := ai.Toy_podshipnika_shest_red_EDT_5.HL;
  AI_Toy_podshipnika_shest_red_EDT_5_LL := ai.Toy_podshipnika_shest_red_EDT_5.LL;
  AI_Toy_podshipnika_shest_red_EDT_5_status := DWORD_TO_UDINT(ai.Toy_podshipnika_shest_red_EDT_5.status);
  AI_Toy_podshipnika_shest_red_EDT_5_value := ai.Toy_podshipnika_shest_red_EDT_5.value;
  AI_Toy_podshipnika_shest_red_EDT_5_HW := ai.Toy_podshipnika_shest_red_EDT_5.HW;
  AI_Toy_podshipnika_shest_red_EDT_5_HA := ai.Toy_podshipnika_shest_red_EDT_5.HA;

  AI_Ty_podshipnika_red_EDT_6_HL := ai.Ty_podshipnika_red_EDT_6.HL;
  AI_Ty_podshipnika_red_EDT_6_LL := ai.Ty_podshipnika_red_EDT_6.LL;
  AI_Ty_podshipnika_red_EDT_6_status := DWORD_TO_UDINT(ai.Ty_podshipnika_red_EDT_6.status);
  AI_Ty_podshipnika_red_EDT_6_value := ai.Ty_podshipnika_red_EDT_6.value;
  AI_Ty_podshipnika_red_EDT_6_HW := ai.Ty_podshipnika_red_EDT_6.HW;
  AI_Ty_podshipnika_red_EDT_6_HA := ai.Ty_podshipnika_red_EDT_6.HA;

  AI_Ty_podshipnika_nagnet_EDT_7_1_HL := ai.Ty_podshipnika_nagnet_EDT_7_1.HL;
  AI_Ty_podshipnika_nagnet_EDT_7_1_LL := ai.Ty_podshipnika_nagnet_EDT_7_1.LL;
  AI_Ty_podshipnika_nagnet_EDT_7_1_status := DWORD_TO_UDINT(ai.Ty_podshipnika_nagnet_EDT_7_1.status);
  AI_Ty_podshipnika_nagnet_EDT_7_1_value := ai.Ty_podshipnika_nagnet_EDT_7_1.value;
  AI_Ty_podshipnika_nagnet_EDT_7_1_HW := ai.Ty_podshipnika_nagnet_EDT_7_1.HW;
  AI_Ty_podshipnika_nagnet_EDT_7_1_HA := ai.Ty_podshipnika_nagnet_EDT_7_1.HA;

  AI_Ty_podshipnika_nagnet_EDT_7_2_HL := ai.Ty_podshipnika_nagnet_EDT_7_2.HL;
  AI_Ty_podshipnika_nagnet_EDT_7_2_LL := ai.Ty_podshipnika_nagnet_EDT_7_2.LL;
  AI_Ty_podshipnika_nagnet_EDT_7_2_status := DWORD_TO_UDINT(ai.Ty_podshipnika_nagnet_EDT_7_2.status);
  AI_Ty_podshipnika_nagnet_EDT_7_2_value := ai.Ty_podshipnika_nagnet_EDT_7_2.value;
  AI_Ty_podshipnika_nagnet_EDT_7_2_HW := ai.Ty_podshipnika_nagnet_EDT_7_2.HW;
  AI_Ty_podshipnika_nagnet_EDT_7_2_HA := ai.Ty_podshipnika_nagnet_EDT_7_2.HA;

  AI_Toy_podshipnika_svobod_konca_EDT_8_1_HL := ai.Toy_podshipnika_svobod_konca_EDT_8_1.HL;
  AI_Toy_podshipnika_svobod_konca_EDT_8_1_LL := ai.Toy_podshipnika_svobod_konca_EDT_8_1.LL;
  AI_Toy_podshipnika_svobod_konca_EDT_8_1_status := DWORD_TO_UDINT(ai.Toy_podshipnika_svobod_konca_EDT_8_1.status);
  AI_Toy_podshipnika_svobod_konca_EDT_8_1_value := ai.Toy_podshipnika_svobod_konca_EDT_8_1.value;
  AI_Toy_podshipnika_svobod_konca_EDT_8_1_HW := ai.Toy_podshipnika_svobod_konca_EDT_8_1.HW;
  AI_Toy_podshipnika_svobod_konca_EDT_8_1_HA := ai.Toy_podshipnika_svobod_konca_EDT_8_1.HA;

  AI_Toy_podshipnika_svobod_konca_EDT_8_2_HL := ai.Toy_podshipnika_svobod_konca_EDT_8_2.HL;
  AI_Toy_podshipnika_svobod_konca_EDT_8_2_LL := ai.Toy_podshipnika_svobod_konca_EDT_8_2.LL;
  AI_Toy_podshipnika_svobod_konca_EDT_8_2_status := DWORD_TO_UDINT(ai.Toy_podshipnika_svobod_konca_EDT_8_2.status);
  AI_Toy_podshipnika_svobod_konca_EDT_8_2_value := ai.Toy_podshipnika_svobod_konca_EDT_8_2.value;
  AI_Toy_podshipnika_svobod_konca_EDT_8_2_HW := ai.Toy_podshipnika_svobod_konca_EDT_8_2.HW;
  AI_Toy_podshipnika_svobod_konca_EDT_8_2_HA := ai.Toy_podshipnika_svobod_konca_EDT_8_2.HA;

  AI_Toy_podshipnika_rab_kol_EDT_9_1_HL := ai.Toy_podshipnika_rab_kol_EDT_9_1.HL;
  AI_Toy_podshipnika_rab_kol_EDT_9_1_LL := ai.Toy_podshipnika_rab_kol_EDT_9_1.LL;
  AI_Toy_podshipnika_rab_kol_EDT_9_1_status := DWORD_TO_UDINT(ai.Toy_podshipnika_rab_kol_EDT_9_1.status);
  AI_Toy_podshipnika_rab_kol_EDT_9_1_value := ai.Toy_podshipnika_rab_kol_EDT_9_1.value;
  AI_Toy_podshipnika_rab_kol_EDT_9_1_HW := ai.Toy_podshipnika_rab_kol_EDT_9_1.HW;
  AI_Toy_podshipnika_rab_kol_EDT_9_1_HA := ai.Toy_podshipnika_rab_kol_EDT_9_1.HA;

  AI_Toy_podshipnika_rab_kol_EDT_9_2_HL := ai.Toy_podshipnika_rab_kol_EDT_9_2.HL;
  AI_Toy_podshipnika_rab_kol_EDT_9_2_LL := ai.Toy_podshipnika_rab_kol_EDT_9_2.LL;
  AI_Toy_podshipnika_rab_kol_EDT_9_2_status := DWORD_TO_UDINT(ai.Toy_podshipnika_rab_kol_EDT_9_2.status);
  AI_Toy_podshipnika_rab_kol_EDT_9_2_value := ai.Toy_podshipnika_rab_kol_EDT_9_2.value;
  AI_Toy_podshipnika_rab_kol_EDT_9_2_HW := ai.Toy_podshipnika_rab_kol_EDT_9_2.HW;
  AI_Toy_podshipnika_rab_kol_EDT_9_2_HA := ai.Toy_podshipnika_rab_kol_EDT_9_2.HA;

  AI_Toy_podshipnika_nerab_kol_EDT_10_1_HL := ai.Toy_podshipnika_nerab_kol_EDT_10_1.HL;
  AI_Toy_podshipnika_nerab_kol_EDT_10_1_LL := ai.Toy_podshipnika_nerab_kol_EDT_10_1.LL;
  AI_Toy_podshipnika_nerab_kol_EDT_10_1_status := DWORD_TO_UDINT(ai.Toy_podshipnika_nerab_kol_EDT_10_1.status);
  AI_Toy_podshipnika_nerab_kol_EDT_10_1_value := ai.Toy_podshipnika_nerab_kol_EDT_10_1.value;
  AI_Toy_podshipnika_nerab_kol_EDT_10_1_HW := ai.Toy_podshipnika_nerab_kol_EDT_10_1.HW;
  AI_Toy_podshipnika_nerab_kol_EDT_10_1_HA := ai.Toy_podshipnika_nerab_kol_EDT_10_1.HA;

  AI_Toy_podshipnika_nerab_kol_EDT_10_2_HL := ai.Toy_podshipnika_nerab_kol_EDT_10_2.HL;
  AI_Toy_podshipnika_nerab_kol_EDT_10_2_LL := ai.Toy_podshipnika_nerab_kol_EDT_10_2.LL;
  AI_Toy_podshipnika_nerab_kol_EDT_10_2_status := DWORD_TO_UDINT(ai.Toy_podshipnika_nerab_kol_EDT_10_2.status);
  AI_Toy_podshipnika_nerab_kol_EDT_10_2_value := ai.Toy_podshipnika_nerab_kol_EDT_10_2.value;
  AI_Toy_podshipnika_nerab_kol_EDT_10_2_HW := ai.Toy_podshipnika_nerab_kol_EDT_10_2.HW;
  AI_Toy_podshipnika_nerab_kol_EDT_10_2_HA := ai.Toy_podshipnika_nerab_kol_EDT_10_2.HA;

  AI_Tholodnogo_vozduha_ED_kanal_1_HL := ai.Tholodnogo_vozduha_ED_kanal_1.HL;
  AI_Tholodnogo_vozduha_ED_kanal_1_LL := ai.Tholodnogo_vozduha_ED_kanal_1.LL;
  AI_Tholodnogo_vozduha_ED_kanal_1_status := DWORD_TO_UDINT(ai.Tholodnogo_vozduha_ED_kanal_1.status);
  AI_Tholodnogo_vozduha_ED_kanal_1_value := ai.Tholodnogo_vozduha_ED_kanal_1.value;
  AI_Tholodnogo_vozduha_ED_kanal_1_HW := ai.Tholodnogo_vozduha_ED_kanal_1.HW;

  AI_Tholodnogo_vozduha_ED_kanal_2_HL := ai.Tholodnogo_vozduha_ED_kanal_2.HL;
  AI_Tholodnogo_vozduha_ED_kanal_2_LL := ai.Tholodnogo_vozduha_ED_kanal_2.LL;
  AI_Tholodnogo_vozduha_ED_kanal_2_status := DWORD_TO_UDINT(ai.Tholodnogo_vozduha_ED_kanal_2.status);
  AI_Tholodnogo_vozduha_ED_kanal_2_value := ai.Tholodnogo_vozduha_ED_kanal_2.value;
  AI_Tholodnogo_vozduha_ED_kanal_2_HW := ai.Tholodnogo_vozduha_ED_kanal_2.HW;

  AI_Tgorjachego_vozduha_ED_kanal_1_HL := ai.Tgorjachego_vozduha_ED_kanal_1.HL;
  AI_Tgorjachego_vozduha_ED_kanal_1_LL := ai.Tgorjachego_vozduha_ED_kanal_1.LL;
  AI_Tgorjachego_vozduha_ED_kanal_1_status := DWORD_TO_UDINT(ai.Tgorjachego_vozduha_ED_kanal_1.status);
  AI_Tgorjachego_vozduha_ED_kanal_1_value := ai.Tgorjachego_vozduha_ED_kanal_1.value;
  AI_Tgorjachego_vozduha_ED_kanal_1_HW := ai.Tgorjachego_vozduha_ED_kanal_1.HW;

  AI_Tgorjachego_vozduha_ED_kanal_2_HL := ai.Tgorjachego_vozduha_ED_kanal_2.HL;
  AI_Tgorjachego_vozduha_ED_kanal_2_LL := ai.Tgorjachego_vozduha_ED_kanal_2.LL;
  AI_Tgorjachego_vozduha_ED_kanal_2_status := DWORD_TO_UDINT(ai.Tgorjachego_vozduha_ED_kanal_2.status);
  AI_Tgorjachego_vozduha_ED_kanal_2_value := ai.Tgorjachego_vozduha_ED_kanal_2.value;
  AI_Tgorjachego_vozduha_ED_kanal_2_HW := ai.Tgorjachego_vozduha_ED_kanal_2.HW;

  AI_Tnarujnogo_vozduha_HL := ai.Tnarujnogo_vozduha.HL;
  AI_Tnarujnogo_vozduha_LL := ai.Tnarujnogo_vozduha.LL;
  AI_Tnarujnogo_vozduha_status := DWORD_TO_UDINT(ai.Tnarujnogo_vozduha.status);
  AI_Tnarujnogo_vozduha_value := ai.Tnarujnogo_vozduha.value;
  AI_Tnarujnogo_vozduha_HW := ai.Tnarujnogo_vozduha.HW;

  AI_Tgaza_na_vhode_H_HL := ai.Tgaza_na_vhode_H.HL;
  AI_Tgaza_na_vhode_H_LL := ai.Tgaza_na_vhode_H.LL;
  AI_Tgaza_na_vhode_H_status := DWORD_TO_UDINT(ai.Tgaza_na_vhode_H.status);
  AI_Tgaza_na_vhode_H_value := ai.Tgaza_na_vhode_H.value;
  AI_Tgaza_na_vhode_H_HW := ai.Tgaza_na_vhode_H.HW;

  AI_Tgaza_na_vyhode_H_HL := ai.Tgaza_na_vyhode_H.HL;
  AI_Tgaza_na_vyhode_H_LL := ai.Tgaza_na_vyhode_H.LL;
  AI_Tgaza_na_vyhode_H_status := DWORD_TO_UDINT(ai.Tgaza_na_vyhode_H.status);
  AI_Tgaza_na_vyhode_H_value := ai.Tgaza_na_vyhode_H.value;
  AI_Tgaza_na_vyhode_H_HW := ai.Tgaza_na_vyhode_H.HW;
  AI_Tgaza_na_vyhode_H_HA := ai.Tgaza_na_vyhode_H.HA;

  AI_Tmasla_do_AVOM_HL := ai.Tmasla_do_AVOM.HL;
  AI_Tmasla_do_AVOM_LL := ai.Tmasla_do_AVOM.LL;
  AI_Tmasla_do_AVOM_status := DWORD_TO_UDINT(ai.Tmasla_do_AVOM.status);
  AI_Tmasla_do_AVOM_value := ai.Tmasla_do_AVOM.value;
  AI_Tmasla_do_AVOM_HW := ai.Tmasla_do_AVOM.HW;

  AI_Tmasla_posle_AVOM_HL := ai.Tmasla_posle_AVOM.HL;
  AI_Tmasla_posle_AVOM_LL := ai.Tmasla_posle_AVOM.LL;
  AI_Tmasla_posle_AVOM_status := DWORD_TO_UDINT(ai.Tmasla_posle_AVOM.status);
  AI_Tmasla_posle_AVOM_value := ai.Tmasla_posle_AVOM.value;
  AI_Tmasla_posle_AVOM_HW := ai.Tmasla_posle_AVOM.HW;

  AI_Tmasla_MB_HL := ai.Tmasla_MB.HL;
  AI_Tmasla_MB_LL := ai.Tmasla_MB.LL;
  AI_Tmasla_MB_status := DWORD_TO_UDINT(ai.Tmasla_MB.status);
  AI_Tmasla_MB_value := ai.Tmasla_MB.value;
  AI_Tmasla_MB_HW := ai.Tmasla_MB.HW;

  AI_Tmasla_MB_TEN_HL := ai.Tmasla_MB_TEN.HL;
  AI_Tmasla_MB_TEN_LL := ai.Tmasla_MB_TEN.LL;
  AI_Tmasla_MB_TEN_status := DWORD_TO_UDINT(ai.Tmasla_MB_TEN.status);
  AI_Tmasla_MB_TEN_value := ai.Tmasla_MB_TEN.value;
  AI_Tmasla_MB_TEN_HW := ai.Tmasla_MB_TEN.HW;

  AI_Tshu_HL := ai.Tshu.HL;
  AI_Tshu_LL := ai.Tshu.LL;
  AI_Tshu_status := DWORD_TO_UDINT(ai.Tshu.status);
  AI_Tshu_value := ai.Tshu.value;

  AI_Pmaslo_sm_nizkoe_HL := ai.Pmaslo_sm_nizkoe.HL;
  AI_Pmaslo_sm_nizkoe_LL := ai.Pmaslo_sm_nizkoe.LL;
  AI_Pmaslo_sm_nizkoe_status := DWORD_TO_UDINT(ai.Pmaslo_sm_nizkoe.status);
  AI_Pmaslo_sm_nizkoe_value := ai.Pmaslo_sm_nizkoe.value;
  AI_Pmaslo_sm_nizkoe_LW := ai.Pmaslo_sm_nizkoe.LW;
  AI_Pmaslo_sm_nizkoe_LA := ai.Pmaslo_sm_nizkoe.LA;

  AI_Pmaslo_sm_vysokoe_HL := ai.Pmaslo_sm_vysokoe.HL;
  AI_Pmaslo_sm_vysokoe_LL := ai.Pmaslo_sm_vysokoe.LL;
  AI_Pmaslo_sm_vysokoe_status := DWORD_TO_UDINT(ai.Pmaslo_sm_vysokoe.status);
  AI_Pmaslo_sm_vysokoe_value := ai.Pmaslo_sm_vysokoe.value;
  AI_Pmaslo_sm_vysokoe_LW := ai.Pmaslo_sm_vysokoe.LW;
  AI_Pmaslo_sm_vysokoe_LA := ai.Pmaslo_sm_vysokoe.LA;

  AI_Pmasla_posle_GNS_HL := ai.Pmasla_posle_GNS.HL;
  AI_Pmasla_posle_GNS_LL := ai.Pmasla_posle_GNS.LL;
  AI_Pmasla_posle_GNS_status := DWORD_TO_UDINT(ai.Pmasla_posle_GNS.status);
  AI_Pmasla_posle_GNS_value := ai.Pmasla_posle_GNS.value;
  AI_Pmasla_posle_GNS_HW := ai.Pmasla_posle_GNS.HW;
  AI_Pmasla_posle_GNS_LW := ai.Pmasla_posle_GNS.LW;

  AI_Pmasla_posle_NU_HL := ai.Pmasla_posle_NU.HL;
  AI_Pmasla_posle_NU_LL := ai.Pmasla_posle_NU.LL;
  AI_Pmasla_posle_NU_status := DWORD_TO_UDINT(ai.Pmasla_posle_NU.status);
  AI_Pmasla_posle_NU_value := ai.Pmasla_posle_NU.value;
  AI_Pmasla_posle_NU_LW := ai.Pmasla_posle_NU.LW;

  AI_Pgaza_na_vhode_nagnetatelia_HL := ai.Pgaza_na_vhode_nagnetatelia.HL;
  AI_Pgaza_na_vhode_nagnetatelia_LL := ai.Pgaza_na_vhode_nagnetatelia.LL;
  AI_Pgaza_na_vhode_nagnetatelia_status := DWORD_TO_UDINT(ai.Pgaza_na_vhode_nagnetatelia.status);
  AI_Pgaza_na_vhode_nagnetatelia_value := ai.Pgaza_na_vhode_nagnetatelia.value;
  AI_Pgaza_na_vhode_nagnetatelia_LW := ai.Pgaza_na_vhode_nagnetatelia.LW;

  AI_Pgaza_na_vyhode_nagnetatelia_HL := ai.Pgaza_na_vyhode_nagnetatelia.HL;
  AI_Pgaza_na_vyhode_nagnetatelia_LL := ai.Pgaza_na_vyhode_nagnetatelia.LL;
  AI_Pgaza_na_vyhode_nagnetatelia_status := DWORD_TO_UDINT(ai.Pgaza_na_vyhode_nagnetatelia.status);
  AI_Pgaza_na_vyhode_nagnetatelia_value := ai.Pgaza_na_vyhode_nagnetatelia.value;
  AI_Pgaza_na_vyhode_nagnetatelia_LW := ai.Pgaza_na_vyhode_nagnetatelia.LW;
  AI_Pgaza_na_vyhode_nagnetatelia_HA := ai.Pgaza_na_vyhode_nagnetatelia.HA;

  AI_Pimpuls_gaz_HL := ai.Pimpuls_gaz.HL;
  AI_Pimpuls_gaz_LL := ai.Pimpuls_gaz.LL;
  AI_Pimpuls_gaz_status := DWORD_TO_UDINT(ai.Pimpuls_gaz.status);
  AI_Pimpuls_gaz_value := ai.Pimpuls_gaz.value;
  AI_Pimpuls_gaz_LW := ai.Pimpuls_gaz.LW;

  AI_dPgaza_na_maslo_filtre_HL := ai.dPgaza_na_maslo_filtre.HL;
  AI_dPgaza_na_maslo_filtre_LL := ai.dPgaza_na_maslo_filtre.LL;
  AI_dPgaza_na_maslo_filtre_status := DWORD_TO_UDINT(ai.dPgaza_na_maslo_filtre.status);
  AI_dPgaza_na_maslo_filtre_value := ai.dPgaza_na_maslo_filtre.value;
  AI_dPgaza_na_maslo_filtre_HW := ai.dPgaza_na_maslo_filtre.HW;

  AI_dPgaza_na_konfuzore_HL := ai.dPgaza_na_konfuzore.HL;
  AI_dPgaza_na_konfuzore_LL := ai.dPgaza_na_konfuzore.LL;
  AI_dPgaza_na_konfuzore_status := DWORD_TO_UDINT(ai.dPgaza_na_konfuzore.status);
  AI_dPgaza_na_konfuzore_value := ai.dPgaza_na_konfuzore.value;
  AI_dPgaza_na_konfuzore_LW := ai.dPgaza_na_konfuzore.LW;

  AI_dPmaslo_gaz_HL := ai.dPmaslo_gaz.HL;
  AI_dPmaslo_gaz_LL := ai.dPmaslo_gaz.LL;
  AI_dPmaslo_gaz_status := DWORD_TO_UDINT(ai.dPmaslo_gaz.status);
  AI_dPmaslo_gaz_value := ai.dPmaslo_gaz.value;
  AI_dPmaslo_gaz_LW := ai.dPmaslo_gaz.LW;
  AI_dPmaslo_gaz_LA := ai.dPmaslo_gaz.LA;

  AI_Os_sdvig_nagnetatelja_plus_HL := ai.Os_sdvig_nagnetatelja_plus.HL;
  AI_Os_sdvig_nagnetatelja_plus_LL := ai.Os_sdvig_nagnetatelja_plus.LL;
  AI_Os_sdvig_nagnetatelja_plus_status := DWORD_TO_UDINT(ai.Os_sdvig_nagnetatelja_plus.status);
  AI_Os_sdvig_nagnetatelja_plus_value := ai.Os_sdvig_nagnetatelja_plus.value;
  AI_Os_sdvig_nagnetatelja_plus_HW := ai.Os_sdvig_nagnetatelja_plus.HW;
  AI_Os_sdvig_nagnetatelja_plus_HA := ai.Os_sdvig_nagnetatelja_plus.HA;

  AI_Os_sdvig_nagnetatelja_minus_HL := ai.Os_sdvig_nagnetatelja_minus.HL;
  AI_Os_sdvig_nagnetatelja_minus_LL := ai.Os_sdvig_nagnetatelja_minus.LL;
  AI_Os_sdvig_nagnetatelja_minus_status := DWORD_TO_UDINT(ai.Os_sdvig_nagnetatelja_minus.status);
  AI_Os_sdvig_nagnetatelja_minus_value := ai.Os_sdvig_nagnetatelja_minus.value;
  AI_Os_sdvig_nagnetatelja_minus_LW := ai.Os_sdvig_nagnetatelja_minus.LW;
  AI_Os_sdvig_nagnetatelja_minus_LA := ai.Os_sdvig_nagnetatelja_minus.LA;

  AI_Yroven_masla_MB_HL := ai.Yroven_masla_MB.HL;
  AI_Yroven_masla_MB_LL := ai.Yroven_masla_MB.LL;
  AI_Yroven_masla_MB_status := DWORD_TO_UDINT(ai.Yroven_masla_MB.status);
  AI_Yroven_masla_MB_value := ai.Yroven_masla_MB.value;
  AI_Yroven_masla_MB_LW := ai.Yroven_masla_MB.LW;

  AI_Kontrol_per_220V_HL := ai.Kontrol_per_220V.HL;
  AI_Kontrol_per_220V_LL := ai.Kontrol_per_220V.LL;
  AI_Kontrol_per_220V_status := DWORD_TO_UDINT(ai.Kontrol_per_220V.status);
  AI_Kontrol_per_220V_value := ai.Kontrol_per_220V.value;
  AI_Kontrol_per_220V_HW := ai.Kontrol_per_220V.HW;
  AI_Kontrol_per_220V_LW := ai.Kontrol_per_220V.LW;

  AI_Kontrol_post_220V_HL := ai.Kontrol_post_220V.HL;
  AI_Kontrol_post_220V_LL := ai.Kontrol_post_220V.LL;
  AI_Kontrol_post_220V_status := DWORD_TO_UDINT(ai.Kontrol_post_220V.status);
  AI_Kontrol_post_220V_value := ai.Kontrol_post_220V.value;
  AI_Kontrol_post_220V_HW := ai.Kontrol_post_220V.HW;
  AI_Kontrol_post_220V_LW := ai.Kontrol_post_220V.LW;

  AI_Tok_statora_HL := ai.Tok_statora.HL;
  AI_Tok_statora_LL := ai.Tok_statora.LL;
  AI_Tok_statora_status := DWORD_TO_UDINT(ai.Tok_statora.status);
  AI_Tok_statora_value := ai.Tok_statora.value;
  AI_Tok_statora_LW := ai.Tok_statora.LW;

  AI_Vibro_skorost_OPED_T1_HL := ai.Vibro_skorost_OPED_T1.HL;
  AI_Vibro_skorost_OPED_T1_LL := ai.Vibro_skorost_OPED_T1.LL;
  AI_Vibro_skorost_OPED_T1_status := DWORD_TO_UDINT(ai.Vibro_skorost_OPED_T1.status);
  AI_Vibro_skorost_OPED_T1_value := ai.Vibro_skorost_OPED_T1.value;
  AI_Vibro_skorost_OPED_T1_HW := ai.Vibro_skorost_OPED_T1.HW;
  AI_Vibro_skorost_OPED_T1_HA := ai.Vibro_skorost_OPED_T1.HA;

  AI_Vibro_skorost_OYPED_T2_HL := ai.Vibro_skorost_OYPED_T2.HL;
  AI_Vibro_skorost_OYPED_T2_LL := ai.Vibro_skorost_OYPED_T2.LL;
  AI_Vibro_skorost_OYPED_T2_status := DWORD_TO_UDINT(ai.Vibro_skorost_OYPED_T2.status);
  AI_Vibro_skorost_OYPED_T2_value := ai.Vibro_skorost_OYPED_T2.value;
  AI_Vibro_skorost_OYPED_T2_HW := ai.Vibro_skorost_OYPED_T2.HW;
  AI_Vibro_skorost_OYPED_T2_HA := ai.Vibro_skorost_OYPED_T2.HA;

  AI_Vibro_skorost_OYP_kolesa_ED_T3_HL := ai.Vibro_skorost_OYP_kolesa_ED_T3.HL;
  AI_Vibro_skorost_OYP_kolesa_ED_T3_LL := ai.Vibro_skorost_OYP_kolesa_ED_T3.LL;
  AI_Vibro_skorost_OYP_kolesa_ED_T3_status := DWORD_TO_UDINT(ai.Vibro_skorost_OYP_kolesa_ED_T3.status);
  AI_Vibro_skorost_OYP_kolesa_ED_T3_value := ai.Vibro_skorost_OYP_kolesa_ED_T3.value;
  AI_Vibro_skorost_OYP_kolesa_ED_T3_HW := ai.Vibro_skorost_OYP_kolesa_ED_T3.HW;
  AI_Vibro_skorost_OYP_kolesa_ED_T3_HA := ai.Vibro_skorost_OYP_kolesa_ED_T3.HA;

  AI_Vibro_skorost_OP_kolesa_RH_T4_HL := ai.Vibro_skorost_OP_kolesa_RH_T4.HL;
  AI_Vibro_skorost_OP_kolesa_RH_T4_LL := ai.Vibro_skorost_OP_kolesa_RH_T4.LL;
  AI_Vibro_skorost_OP_kolesa_RH_T4_status := DWORD_TO_UDINT(ai.Vibro_skorost_OP_kolesa_RH_T4.status);
  AI_Vibro_skorost_OP_kolesa_RH_T4_value := ai.Vibro_skorost_OP_kolesa_RH_T4.value;
  AI_Vibro_skorost_OP_kolesa_RH_T4_HW := ai.Vibro_skorost_OP_kolesa_RH_T4.HW;
  AI_Vibro_skorost_OP_kolesa_RH_T4_HA := ai.Vibro_skorost_OP_kolesa_RH_T4.HA;

  AI_Vibro_skorost_OP_shesterni_RED_T5_HL := ai.Vibro_skorost_OP_shesterni_RED_T5.HL;
  AI_Vibro_skorost_OP_shesterni_RED_T5_LL := ai.Vibro_skorost_OP_shesterni_RED_T5.LL;
  AI_Vibro_skorost_OP_shesterni_RED_T5_status := DWORD_TO_UDINT(ai.Vibro_skorost_OP_shesterni_RED_T5.status);
  AI_Vibro_skorost_OP_shesterni_RED_T5_value := ai.Vibro_skorost_OP_shesterni_RED_T5.value;
  AI_Vibro_skorost_OP_shesterni_RED_T5_HW := ai.Vibro_skorost_OP_shesterni_RED_T5.HW;
  AI_Vibro_skorost_OP_shesterni_RED_T5_HA := ai.Vibro_skorost_OP_shesterni_RED_T5.HA;

  AI_Vibro_skorost_OP_shesterni_RED_T6_HL := ai.Vibro_skorost_OP_shesterni_RED_T6.HL;
  AI_Vibro_skorost_OP_shesterni_RED_T6_LL := ai.Vibro_skorost_OP_shesterni_RED_T6.LL;
  AI_Vibro_skorost_OP_shesterni_RED_T6_status := DWORD_TO_UDINT(ai.Vibro_skorost_OP_shesterni_RED_T6.status);
  AI_Vibro_skorost_OP_shesterni_RED_T6_value := ai.Vibro_skorost_OP_shesterni_RED_T6.value;
  AI_Vibro_skorost_OP_shesterni_RED_T6_HW := ai.Vibro_skorost_OP_shesterni_RED_T6.HW;
  AI_Vibro_skorost_OP_shesterni_RED_T6_HA := ai.Vibro_skorost_OP_shesterni_RED_T6.HA;
END_FUNCTION_BLOCK

FUNCTION TwoUint_To_UDINT : UDINT
  VAR_INPUT
    val1 : UINT;
    val2 : UINT;
  END_VAR

  TwoUint_To_UDINT:= DWORD_TO_UDINT(UINT_TO_DWORD(val1) OR shl(UINT_TO_DWORD(val2), 16));
END_FUNCTION

FUNCTION_BLOCK proc_DI
  VAR
    di_0 : fb_DiSourceMlp;
    di_1 : fb_DiSourceMlp;
    di_2 : fb_DiSourceMlp;
    di_3 : fb_DiSourceMlp;
    di_4 : fb_DiSourceMlp;
    di_5 : fb_DiSourceMlp;
    di_6 : fb_DiSourceMlp;
    di_7 : fb_DiSourceMlp;
    di_8 : fb_DiSourceMlp;
    di_9 : fb_DiSourceMlp;
    di_10 : fb_DiSourceMlp;
    di_11 : fb_DiSourceMlp;
    di_12 : fb_DiSourceMlp;
    di_13 : fb_DiSourceMlp;
    di_14 : fb_DiSourceMlp;
    di_15 : fb_DiSourceMlp;
    di_16 : fb_DiSourceMlp;
    di_17 : fb_DiSourceMlp;
    di_18 : fb_DiSourceMlp;
    di_19 : fb_DiSourceMlp;
    di_20 : fb_DiSourceMlp;
    di_21 : fb_DiSourceMlp;
  END_VAR
  VAR_EXTERNAL
    arDIN_0 : TItemDIN;
    arDIN_1 : TItemDIN;
    arDIN_2 : TItemDIN;
    arDIN_3 : TItemDIN;
    arDIN_4 : TItemDIN;
    arDIN_5 : TItemDIN;
    arDIN_6 : TItemDIN;
    arDIN_7 : TItemDIN;
    arDIN_8 : TItemDIN;
    arDIN_9 : TItemDIN;
    arDIN_10 : TItemDIN;
    arDIN_11 : TItemDIN;
    arDIN_12 : TItemDIN;
    arDIN_13 : TItemDIN;
    arDIN_14 : TItemDIN;
    arDIN_15 : TItemDIN;
    arDIN_16 : TItemDIN;
    arDIN_17 : TItemDIN;
    arDIN_18 : TItemDIN;
    arDIN_19 : TItemDIN;
    arDIN_20 : TItemDIN;
    arDIN_21 : TItemDIN;
    di : DiConfig;
    DI_0_1_wValue : UDINT;
    DI_10_11_wValue : UDINT;
    DI_12_13_wValue : UDINT;
    DI_14_15_wValue : UDINT;
    DI_16_17_wValue : UDINT;
    DI_18_19_wValue : UDINT;
    DI_20_21_wValue : UDINT;
    DI_2_3_wValue : UDINT;
    DI_4_5_wValue : UDINT;
    DI_6_7_wValue : UDINT;
    DI_8_9_wValue : UDINT;
    A1_12_err_mode : UINT;
    A1_13_err_mode : UINT;
    A1_14_err_mode : UINT;
    A1_15_err_mode : UINT;
    A2_10_err_mode : UINT;
    A2_4_err_mode : UINT;
    A2_5_err_mode : UINT;
    A2_6_err_mode : UINT;
    A2_7_err_mode : UINT;
    A2_8_err_mode : UINT;
    A2_9_err_mode : UINT;
    arERR_11 : TItemDIN;
    arERR_12 : TItemDIN;
    arERR_13 : TItemDIN;
    arERR_14 : TItemDIN;
    arERR_18 : TItemDIN;
    arERR_19 : TItemDIN;
    arERR_20 : TItemDIN;
    arERR_21 : TItemDIN;
    arERR_22 : TItemDIN;
    arERR_23 : TItemDIN;
    arERR_24 : TItemDIN;
  END_VAR

  (* Циклический опрос. Входные дискретные параметры *)
  (* Модуль A1-12 *)
  di_0(arDIN := arDIN_0, strDI:=di.di_0, err_mod:=arERR_11);
  di_1(arDIN := arDIN_1, strDI:=di.di_1, err_mod:=arERR_11);
  DI_0_1_wValue:=TwoUint_To_UDINT(arDIN_0.wValue, arDIN_1.wValue);
  A1_12_err_mode:= arERR_11.wValue;

  (* Модуль A1-13 *)
  di_2(arDIN := arDIN_2, strDI:=di.di_2,  err_mod:=arERR_12);
  di_3(arDIN := arDIN_3, strDI:=di.di_3,  err_mod:=arERR_12);
  DI_2_3_wValue:=TwoUint_To_UDINT(arDIN_2.wValue, arDIN_3.wValue);
  A1_13_err_mode:= arERR_12.wValue;

  (* Модуль A1-14 *)
  di_4(arDIN := arDIN_4, strDI:=di.di_4,  err_mod:=arERR_13);
  di_5(arDIN := arDIN_5, strDI:=di.di_5,  err_mod:=arERR_13);
  DI_4_5_wValue:=TwoUint_To_UDINT(arDIN_4.wValue, arDIN_5.wValue);
  A1_14_err_mode:= arERR_13.wValue;

  (* Модуль A1-15 *)
  di_6(arDIN := arDIN_6, strDI:=di.di_6,  err_mod:=arERR_14);
  di_7(arDIN := arDIN_7, strDI:=di.di_7,  err_mod:=arERR_14);
  DI_6_7_wValue:=TwoUint_To_UDINT(arDIN_6.wValue, arDIN_7.wValue);
  A1_15_err_mode:= arERR_14.wValue;

  (* Модуль A2-4 *)
  di_8(arDIN := arDIN_8, strDI:=di.di_8,  err_mod:=arERR_18);
  di_9(arDIN := arDIN_9, strDI:=di.di_9,  err_mod:=arERR_18);
  DI_8_9_wValue:=TwoUint_To_UDINT(arDIN_8.wValue, arDIN_9.wValue);
  A2_4_err_mode:= arERR_18.wValue;

  (* Модуль A2-5 *)
  di_10(arDIN := arDIN_10, strDI:=di.di_10,  err_mod:=arERR_19);
  di_11(arDIN := arDIN_11, strDI:=di.di_11,  err_mod:=arERR_19);
  DI_10_11_wValue:=TwoUint_To_UDINT(arDIN_10.wValue, arDIN_11.wValue);
  A2_5_err_mode:= arERR_19.wValue;

  (* Модуль A2-6 *)
  di_12(arDIN := arDIN_12, strDI:=di.di_12,  err_mod:=arERR_20);
  di_13(arDIN := arDIN_13, strDI:=di.di_13,  err_mod:=arERR_20);
  DI_12_13_wValue:=TwoUint_To_UDINT(arDIN_12.wValue, arDIN_13.wValue);
  A2_6_err_mode:= arERR_20.wValue;

  (* Модуль A2-7 *)
  di_14(arDIN := arDIN_14, strDI:=di.di_14,  err_mod:=arERR_21);
  di_15(arDIN := arDIN_15, strDI:=di.di_15,  err_mod:=arERR_21);
  DI_14_15_wValue:=TwoUint_To_UDINT(arDIN_14.wValue, arDIN_15.wValue);
  A2_7_err_mode:= arERR_21.wValue;

  di_16(arDIN := arDIN_16, strDI:=di.di_16,  err_mod:=arERR_22);
  di_17(arDIN := arDIN_17, strDI:=di.di_17,  err_mod:=arERR_22);
  DI_16_17_wValue:=TwoUint_To_UDINT(arDIN_16.wValue, arDIN_17.wValue);
  A2_8_err_mode:= arERR_22.wValue;

  di_18(arDIN := arDIN_18, strDI:=di.di_18,  err_mod:=arERR_23);
  di_19(arDIN := arDIN_19, strDI:=di.di_19,  err_mod:=arERR_23);
  DI_18_19_wValue:=TwoUint_To_UDINT(arDIN_18.wValue, arDIN_19.wValue);
  A2_9_err_mode:= arERR_23.wValue;

  di_20(arDIN := arDIN_20, strDI:=di.di_20,  err_mod:=arERR_24);
  di_21(arDIN := arDIN_21, strDI:=di.di_21,  err_mod:=arERR_24);
  DI_20_21_wValue:=TwoUint_To_UDINT(arDIN_20.wValue, arDIN_21.wValue);
  A2_10_err_mode:= arERR_24.wValue;
END_FUNCTION_BLOCK

FUNCTION_BLOCK proc_AO_Init
  VAR_INPUT
    init : BOOL;
  END_VAR
  VAR
    stAO_Ini : fb_AO_Init;
    inits : UINT;
  END_VAR
  VAR_INPUT
    initiales : UINT;
  END_VAR
  VAR_EXTERNAL
    ao : AOConfig;
  END_VAR

  (* Инициализация начало. Входные аналоговые параметры *)

  inits := 0; (* Флаг необходимости инициализации структур-дескрипторов *)

  (* Модуль A10 *)
  (* [A10, AO0] Резерв (A) *)
  stAO_Ini(data_Ini := TRUE, (*outLL := 4000.0, outHL := 20000.0,*)
    newLL_ISVALIDREF := TRUE, newHL_ISVALIDREF := TRUE,
    newLL := 0.0, newHL := 100.0,
    strAO := ao.Reserv_AO_1);
  inits := inits + BOOL_TO_UINT(stAO_Ini.Init);

  (* [A1-10, AO1] Резерв (A) *)
  stAO_Ini(data_Ini := TRUE, (*outLL := 4000.0, outHL := 20000.0,*)
    (*newLL_ISVALIDREF := TRUE, newHL_ISVALIDREF := TRUE,*)
    (*newLL := 0.0, newHL := 100.0,*)
  strAO := ao.Reserv_AO_2);
  inits := inits + BOOL_TO_UINT(stAO_Ini.Init);

  initiales := 0;
  IF init THEN initiales := inits; END_IF;
END_FUNCTION_BLOCK

FUNCTION_BLOCK fb_Timings
  VAR_EXTERNAL CONSTANT
    req_Cycle : REAL;
  END_VAR
  VAR_EXTERNAL
    gF_T_100mSec : BOOL;
    gT_1Sec : BOOL;
    gF_T_1Sec : BOOL;
    gT_1Min : BOOL;
    gR_T_1Min : BOOL;
    gF_T_1Min : BOOL;
    del_T : REAL;
    cur_Cycle : REAL;
  END_VAR
  VAR
    Tmr_100_ms : REAL;
  END_VAR
  VAR_EXTERNAL
    T_1SEC : REAL;
  END_VAR
  VAR
    Tmr_1_s : REAL;
    Tmr_1_min : REAL;
  END_VAR

  (* Обработка времени. *)
  Tmr_100_ms := Tmr_100_ms + cur_Cycle;
  gF_T_100mSec := FALSE;
  IF Tmr_100_ms >= 0.1 THEN Tmr_100_ms := 0.0; gF_T_100mSec := TRUE; END_IF;

  Tmr_1_s := Tmr_1_s + cur_Cycle;
  gF_T_1Sec := FALSE;
  IF Tmr_1_s >= 1.0 THEN Tmr_1_s := 0.0; gF_T_1Sec := TRUE; END_IF;

  T_1SEC := T_1SEC + cur_Cycle;
  gT_1Sec := FALSE;
  IF T_1SEC >= 2.0 THEN T_1SEC := 0.0;
    ELSIF T_1SEC >= 1.0 THEN gT_1Sec := TRUE; END_IF;

  IF Tmr_1_min > 60.0 THEN
      Tmr_1_min := 0.0; gF_T_1Min := gT_1Min; gT_1Min := NOT gT_1Min; gR_T_1Min := gT_1Min;
    ELSE
      Tmr_1_min := Tmr_1_min + cur_Cycle; gR_T_1Min := FALSE; gF_T_1Min := FALSE;
  END_IF;
  del_T:= cur_Cycle;
END_FUNCTION_BLOCK

FUNCTION autoRunProtections : BOOL
  VAR_IN_OUT
    protections : ProtectionsConfig;
  END_VAR

  runAiProtection(protections.Topornogo_podshipnika_EDT_1);

      runAiProtection(protections.Toy_podshipnika_EDT_2);

      runAiProtection(protections.Toy_podshipnika_kol_EDT_3);

      runAiProtection(protections.Toy_podshipnika_kol_EDT_4);

      runAiProtection(protections.To_podshipnika_shest_red_EDT_5);

      runAiProtection(protections.To_podshipnika_shest_red_EDT_6);

      runAiProtection(protections.To_podshipnika_N_EDT_7);

      runAiProtection(protections.To_podshipnika_svob_konca_EDT_8);

      runAiProtection(protections.Ty_podshipnika_rab_kol_EDT_9);

      runAiProtection(protections.Typornogo_podshipnika_nerab_kolodok_HT_10);

      runAiProtection(protections.Tgaza_na_vyhode_H);

      runAiProtection(protections.Os_sdvig_nagnetatelja_plus);

      runAiProtection(protections.Os_sdvig_nagnetatelja_minus);

      runAiProtection(protections.Pgaza_na_vyhode_nagnetatelia_GPA_STOP);

      runAiProtection(protections.Pgaza_na_vhode_nagnetatelia_GPA_STOP);

      runAiProtection(protections.Pgaza_na_vyhode_nagnetatelia);

      runAiProtection(protections.dPmaslo_gaz);

      runAiProtection(protections.Pmaslo_sm_nizkoe);

      runAiProtection(protections.Pmaslo_sm_vysokoe);

      runAiProtection(protections.Vibro_skorost_OPED_T1);

      runAiProtection(protections.Vibro_skorost_OPED_T2);

      runAiProtection(protections.Vibro_skorost_OYP_kolesa_ED_T3);

      runAiProtection(protections.Vibro_skorost_OP_kolesa_RH_T4);

      runAiProtection(protections.Vibro_skorost_OP_shesterni_RED_T5);

      runAiProtection(protections.Vibro_skorost_OP_shesterni_RED_T6);

      runDiProtection(protections.dPmaslo_gaz_less100);

      runDiProtection(protections.AO_PRU);

      runDiProtection(protections.Reg_vozb_off);

      runDiProtection(protections.Fail_chastotnii_pusk);

      runDiProtection(protections.AOKC_SHKC);

      runDiProtection(protections.mvOff);

      runDiProtection(protections.AO_ot_SHU);

      runDiProtection(protections.Off_avar_vikluchatel);

      runDiProtection(protections.Kran1_sdvig);

      runDiProtection(protections.Kran2_sdvig);
END_FUNCTION

FUNCTION runAllProtections : BOOL
  VAR_IN_OUT
    protections : ProtectionsConfig;
  END_VAR

  runAiProtection(protections.Topornogo_podshipnika_EDT_1);
  runAiProtection(protections.Toy_podshipnika_EDT_2);
  runAiProtection(protections.Toy_podshipnika_kol_EDT_3);
  runAiProtection(protections.Toy_podshipnika_kol_EDT_4);
  runAiProtection(protections.To_podshipnika_shest_red_EDT_5);
  runAiProtection(protections.To_podshipnika_shest_red_EDT_6);
  runAiProtection(protections.To_podshipnika_N_EDT_7);
  runAiProtection(protections.To_podshipnika_svob_konca_EDT_8);
  runAiProtection(protections.Ty_podshipnika_rab_kol_EDT_9);
  runAiProtection(protections.Typornogo_podshipnika_nerab_kolodok_HT_10);
  runAiProtection(protections.Tgaza_na_vyhode_H);
  runAiProtection(protections.Os_sdvig_nagnetatelja_plus);
  runAiProtection(protections.Os_sdvig_nagnetatelja_minus);
  runAiProtection(protections.Pgaza_na_vyhode_nagnetatelia_GPA_STOP);
  runAiProtection(protections.Pgaza_na_vhode_nagnetatelia_GPA_STOP);
  runAiProtection(protections.Pgaza_na_vyhode_nagnetatelia);
  runAiProtection(protections.dPmaslo_gaz);
  runAiProtection(protections.Pmaslo_sm_nizkoe);
  runAiProtection(protections.Pmaslo_sm_vysokoe);
  runAiProtection(protections.Vibro_skorost_OPED_T1);
  runAiProtection(protections.Vibro_skorost_OPED_T2);
  runAiProtection(protections.Vibro_skorost_OYP_kolesa_ED_T3);
  runAiProtection(protections.Vibro_skorost_OP_kolesa_RH_T4);
  runAiProtection(protections.Vibro_skorost_OP_shesterni_RED_T5);
  runAiProtection(protections.Vibro_skorost_OP_shesterni_RED_T6);
